    //=========================================================================
    // TRK_COMPLETE
    // Kết thúc một object; nếu Execute còn TRUE thì tìm object tiếp theo.
    //=========================================================================
    E_TrackingState.TRK_COMPLETE:

        // Chu trình một object đã hoàn thành.
		Runtime.Response.Busy := FALSE;
		Runtime.Response.Done := TRUE;
	
		// Giữ output ở trạng thái an toàn.
		VacuumCommand := FALSE;
		BlowCommand := FALSE;
	
		// Chỉ về IDLE khi tầng Command Engine hạ Execute.
		IF NOT Execute THEN
			Runtime.Response.Accepted := FALSE;
			Runtime.Response.Done := FALSE;
			Runtime.State := E_TrackingState.TRK_IDLE;
		END_IF;


    //=========================================================================
    // TRK_ABORT_ACTIVE
    // Hủy motion vì object vượt vùng trước khi VacuumOK.
    //=========================================================================
    E_TrackingState.TRK_ABORT_ACTIVE:

        // Tắt hút vì chưa giữ được vật.
        VacuumCommand := FALSE;

        // Tắt thổi.
        BlowCommand := FALSE;

        // Bật yêu cầu abort motion.
        MotionAbort := TRUE;

        // Khi Motion Manager xác nhận abort hoàn tất.
        IF MotionAbortDone THEN
            // Hạ yêu cầu abort.
            MotionAbort := FALSE;

            // Xóa trạng thái motion.
            xMotionIssued := FALSE;
            xMotionRequestPending := FALSE;
            xMotionActive := FALSE;

            // Nếu PCS không còn InUse thì có thể tắt tracking.
            IF NOT fbTrackBelt.InUse THEN
                xTrackExecute := FALSE;

                // Chuyển sang vị trí an toàn.
                Runtime.State := E_TrackingState.TRK_MOVE_SAFE;
            END_IF;
        END_IF;

    //=========================================================================
    // TRK_MOVE_SAFE
    // Đưa robot về LeavePos sau khi bỏ object.
    //=========================================================================
    E_TrackingState.TRK_MOVE_SAFE:

        // Tắt hút.
        VacuumCommand := FALSE;

        // Tạo request Move Safe.
        IF NOT xMotionIssued AND NOT xMotionRequestPending AND NOT xMotionActive THEN

            // Dùng LeavePos làm điểm an toàn.
            MotionTarget := Config.LeavePos;

            // Dùng thông số Leave.
            MotionSpeed := Config.Motion.Leave.Speed;

            MotionAcceleration := Config.Motion.Leave.Acceleration;

            MotionDeceleration := Config.Motion.Leave.Deceleration;

            MotionJerk := Config.Motion.Leave.Jerk;

            MotionBlendRadius := Config.Motion.Leave.BlendRadius;

            // Chạy trong hệ robot/base.
            MotionCoordSystem := E_AppCoordSystem.APP_COORD_ROBOT_BASE;

            // Mã lệnh MoveL.
            MotionCommand := 2;

            // Bật request pending.
            xMotionRequestPending := TRUE;

            // Đánh dấu đã tạo lệnh.
            xMotionIssued := TRUE;
        END_IF;

        // Adapter đã nhận request.
        IF MotionAccepted AND xMotionRequestPending THEN
            xMotionRequestPending := FALSE;
            xMotionActive := TRUE;
        END_IF;

        // Move Safe hoàn thành.
        IF MotionDone AND xMotionActive THEN
            xMotionActive := FALSE;
            xMotionIssued := FALSE;

            Runtime.State := E_TrackingState.TRK_RELEASE_OBJECT;

        // Move Safe lỗi.
        ELSIF MotionError AND xMotionActive THEN
            xMotionActive := FALSE;

            Runtime.Response.Error := TRUE;
            Runtime.Response.ErrorID := MotionErrorID;

            Runtime.State := E_TrackingState.TRK_ERROR;
        END_IF;

    //=========================================================================
    // TRK_RELEASE_OBJECT
    // Giải phóng object MISSED và tiếp tục object kế tiếp.
    //=========================================================================
    E_TrackingState.TRK_RELEASE_OBJECT:

        // Tắt hút.
        VacuumCommand := FALSE;

        // Chỉ release khi PCS không còn InUse.
        IF NOT fbTrackBelt.InUse THEN
            // Tắt tracking PCS.
            xTrackExecute := FALSE;

            // Kiểm tra index trước khi truy cập Queue.
            IF Runtime.SelectedObjectIndex >= 1 AND Runtime.SelectedObjectIndex <= GVL.C_MAX_TRACK_OBJECTS THEN

                // Giải phóng object.
                Queue.Objects[Runtime.SelectedObjectIndex].Reserved := FALSE;
            END_IF;

            // Giải phóng ActiveIndex.
            Queue.ActiveIndex := GVL.C_INVALID_INDEX;

            // Xóa object active trong Runtime.
            Runtime.SelectedObjectIndex := 0;
            Runtime.SelectedObjectID := 0;

            // Xóa thông tin PCS.
            Runtime.PCSInfo.Valid := FALSE;
            Runtime.PCSInfo.InUse := FALSE;

            // Xóa trạng thái tool.
            xVacuumCaptured := FALSE;

            // Xóa trạng thái motion.
            xMotionIssued := FALSE;
            xMotionRequestPending := FALSE;
            xMotionActive := FALSE;

            // Tiếp tục tìm object khác.
            Runtime.State := E_TrackingState.TRK_FIND_OBJECT;
        END_IF;

    //=========================================================================
    // TRK_ABORTING
    // Hủy toàn ứng dụng khi Execute bị hạ.
    //=========================================================================
    E_TrackingState.TRK_ABORTING:

        // Tắt hút.
        VacuumCommand := FALSE;

        // Tắt thổi.
        BlowCommand := FALSE;

        // Yêu cầu abort motion.
        MotionAbort := TRUE;

        // Nếu có object active thì đánh dấu ABORTED.
        IF Runtime.SelectedObjectIndex >= 1 AND Runtime.SelectedObjectIndex <= GVL.C_MAX_TRACK_OBJECTS THEN

            Queue.Objects[Runtime.SelectedObjectIndex].State := E_TrackingObjectState.OBJ_ABORTED;

            Queue.Objects[Runtime.SelectedObjectIndex].Reserved := FALSE;
        END_IF;

        // Khi abort motion xong và PCS không còn InUse.
        IF MotionAbortDone AND NOT fbTrackBelt.InUse THEN

            // Hạ abort.
            MotionAbort := FALSE;

            // Tắt tracking PCS.
            xTrackExecute := FALSE;

            // Giải phóng ActiveIndex.
            Queue.ActiveIndex := GVL.C_INVALID_INDEX;

            // Xóa object active.
            Runtime.SelectedObjectIndex := 0;
            Runtime.SelectedObjectID := 0;

            // Xóa Busy và Accepted.
            Runtime.Response.Busy := FALSE;
            Runtime.Response.Accepted := FALSE;

            // Về IDLE.
            Runtime.State := E_TrackingState.TRK_IDLE;
        END_IF;

    //=========================================================================
    // TRK_ERROR
    // Giữ lỗi để Application Manager/HMI đọc.
    //=========================================================================
    E_TrackingState.TRK_ERROR:

        // Manager không còn xử lý bình thường.
        Runtime.Response.Busy := FALSE;

        // Giữ cờ Error.
        Runtime.Response.Error := TRUE;

        // Tắt hút.
        VacuumCommand := FALSE;

        // Tắt thổi.
        BlowCommand := FALSE;

        // Yêu cầu abort motion.
        MotionAbort := TRUE;

        // Nếu có object active thì đánh dấu ERROR.
        IF Runtime.SelectedObjectIndex >= 1 AND Runtime.SelectedObjectIndex <= GVL.C_MAX_TRACK_OBJECTS THEN

            Queue.Objects[Runtime.SelectedObjectIndex].State := E_TrackingObjectState.OBJ_ERROR;

            Queue.Objects[Runtime.SelectedObjectIndex].Reserved := FALSE;
        END_IF;

        // Chỉ tắt tracking khi PCS không còn InUse.
        IF NOT fbTrackBelt.InUse THEN
            xTrackExecute := FALSE;
        END_IF;

    //=========================================================================
    // STATE KHÔNG HỢP LỆ
    //=========================================================================
    ELSE
        // Báo lỗi state không hợp lệ.
        Runtime.Response.Error := TRUE;

        // Mã lỗi nội bộ cho state không hợp lệ.
        Runtime.Response.ErrorID := 6999;

        // Chuyển về TRK_ERROR.
        Runtime.State := E_TrackingState.TRK_ERROR;

END_CASE;

END_FUNCTION_BLOCK

// Just_Motion_Control_x86_64_Linux_SM_WV/Application/FB_/TOOL/FB_ToolManager
FUNCTION_BLOCK FB_ToolManager
VAR_INPUT

    // Cho phép Tool Manager.
    Enable : BOOL;

    // Command hiện tại.
    Command : ST_ToolCommand;

    // Cấu hình Tool.
    Config : ST_ToolConfig;

END_VAR

VAR_IN_OUT

    // Runtime Status của Tool.
    Status : ST_ToolStatus;

END_VAR

VAR

    // Bắt cạnh lên của Execute.
    rtExecute : R_TRIG;

    // Lệnh Tool đang chạy.
    eActiveCommand : E_ToolCommandType;

    // Timer dùng khi không cấu hình DI.
    tonAction : TON;

    // Timer giới hạn thời gian lệnh Tool.
    tonTimeout : TON;

    // Timer xác nhận GripOK ổn định.
    tonConfirm : TON;

    // Điều kiện lệnh Tool hoàn thành.
    xActionOK : BOOL;

    // Giá trị DI đang kiểm tra.
    xFeedbackDI : BOOL;

    // Thời gian giả lập nếu không có Sensor.
    tAction : TIME;

    // Timeout của lệnh Tool.
    tTimeout : TIME;

END_VAR

(*
===============================================================================
FUNCTION BLOCK
    FB_ToolManager

DESCRIPTION
    Điều khiển một Tool độc lập.

SUPPORTED COMMANDS
    - DOWN
    - GRIP
    - UP
    - RELEASE

FEEDBACK RULE
    - Nếu DI Channel > 0:
          Dùng DI làm điều kiện hoàn thành.
    - Nếu DI Channel = 0:
          Dùng Timer cấu hình tương ứng.
    - Nếu UseUpDown = FALSE:
          DOWN và UP hoàn thành ngay.

IMPORTANT
    - Chỉ FB này được phép ghi request IO của Tool.
    - Interpreter không nên ghi trực tiếp vào các DO đã thuộc Tool.
===============================================================================
*)

//=============================================================================
// DEFAULT PULSE OUTPUTS
//=============================================================================
Status.Accepted := FALSE;
Status.Done := FALSE;


//=============================================================================
// COPY TOOL ID TO STATUS
//=============================================================================
Status.ToolID := Config.ToolID;


//=============================================================================
// RESET / DISABLE
//=============================================================================
IF NOT Enable OR Command.Reset THEN

    Status.Busy := FALSE;

    Status.Error := FALSE;
    Status.ErrorID := 0;

    Status.State :=
        E_ToolRuntimeState.IDLE;

    tonAction(IN := FALSE);
    tonTimeout(IN := FALSE);
    tonConfirm(IN := FALSE);

    RETURN;

END_IF;


//=============================================================================
// ABORT
//=============================================================================
IF Command.Abort THEN

    Status.Busy := FALSE;

    Status.Error := TRUE;
    Status.ErrorID := 9299;

    Status.State :=
        E_ToolRuntimeState.ERROR;

    RETURN;

END_IF;


//=============================================================================
// DETECT NEW COMMAND
//=============================================================================
rtExecute(CLK := Command.Execute);

IF rtExecute.Q AND NOT Status.Busy THEN

    // Lưu loại lệnh hiện tại.
    eActiveCommand :=
        Command.CommandType;

    // Handshake.
    Status.Accepted := TRUE;
    Status.Busy := TRUE;

    Status.Error := FALSE;
    Status.ErrorID := 0;

    Status.ResponseCommandID :=
        Command.CommandID;

    // Reset timer trước khi bắt đầu lệnh mới.
    tonAction(IN := FALSE);
    tonTimeout(IN := FALSE);
    tonConfirm(IN := FALSE);

    // Gán State runtime.
    CASE eActiveCommand OF

        E_ToolCommandType.DOWN:
            Status.State :=
                E_ToolRuntimeState.DOWNING;

        E_ToolCommandType.GRIP:
            Status.State :=
                E_ToolRuntimeState.GRIPPING;

        E_ToolCommandType.UP:
            Status.State :=
                E_ToolRuntimeState.UPPING;

        E_ToolCommandType.RELEASE:
            Status.State :=
                E_ToolRuntimeState.RELEASING;

        ELSE
            Status.Busy := FALSE;
            Status.Done := TRUE;

    END_CASE;

END_IF;


//=============================================================================
// NO ACTIVE COMMAND
//=============================================================================
IF NOT Status.Busy THEN
    RETURN;
END_IF;


//=============================================================================
// RESET LOCAL ACTION FLAGS
//=============================================================================
xActionOK := FALSE;
xFeedbackDI := FALSE;

tAction := T#0MS;
tTimeout := T#1S;


//=============================================================================
// EXECUTE ACTIVE COMMAND
//=============================================================================
CASE eActiveCommand OF


    //=========================================================================
    // ACTION: DOWN
    //=========================================================================
    E_ToolCommandType.DOWN:

        // Tool không có cơ cấu Up/Down.
        IF NOT Config.UseUpDown THEN

            xActionOK := TRUE;

        ELSE

            //-----------------------------------------------------------------
            // COMMAND DOWN OUTPUT
            //-----------------------------------------------------------------
			
			IF Config.IO.UseSingleUpDownDO THEN
				// Single DO: phat muc DOWN.
				IF Config.IO.UpDownDOChannel > 0 AND Config.IO.UpDownDOChannel <= GVL.C_MAX_DO THEN
					GVL.Y[Config.IO.UpDownDOChannel] := Config.IO.DownDOActiveLevel;
				END_IF;
			ELSE
				// Dual DO: bat Down, tat Up.
				IF Config.IO.DownDOChannel > 0 AND Config.IO.DownDOChannel <= GVL.C_MAX_DO THEN
					GVL.Y[Config.IO.DownDOChannel] := Config.IO.DownDOActiveLevel;
				END_IF;
			
				IF Config.IO.UpDOChannel > 0 AND Config.IO.UpDOChannel <= GVL.C_MAX_DO THEN
					GVL.Y[Config.IO.UpDOChannel] := NOT Config.IO.UpDOActiveLevel;
				END_IF;
			END_IF;


            //-----------------------------------------------------------------
            // CHECK DOWN FEEDBACK
            //-----------------------------------------------------------------
            IF Config.IO.DownOKDIChannel = 0 THEN

                // Không có DI -> dùng Timer.
                tAction :=
                    Config.DownTimeNoSensor;

                tonAction(
                    IN := TRUE,
                    PT := tAction
                );

                xActionOK :=
                    tonAction.Q;

            ELSE

                // Có DI -> dùng Sensor.
                xActionOK :=
                    GVL.X[
                        Config.IO.DownOKDIChannel
                    ] = Config.IO.DownOKDIActiveLevel;

            END_IF;


            // Timeout của DOWN.
            tTimeout :=
                Config.DownTimeout;

        END_IF;


    //=========================================================================
    // ACTION: GRIP
    //=========================================================================
    E_ToolCommandType.GRIP:

        //---------------------------------------------------------------------
        // RESET RELEASE OUTPUT
        //---------------------------------------------------------------------
        IF Config.IO.UseSingleGripReleaseDO THEN
			IF Config.IO.GripReleaseDOChannel > 0 AND Config.IO.GripReleaseDOChannel <= GVL.C_MAX_DO THEN
				GVL.Y[Config.IO.GripReleaseDOChannel] := Config.IO.GripDOActiveLevel;
			END_IF;
		ELSE
			IF Config.IO.ReleaseDOChannel > 0 AND Config.IO.ReleaseDOChannel <= GVL.C_MAX_DO THEN
				GVL.Y[Config.IO.ReleaseDOChannel] := NOT Config.IO.ReleaseDOActiveLevel;
			END_IF;
			IF Config.IO.GripDOChannel > 0 AND Config.IO.GripDOChannel <= GVL.C_MAX_DO THEN
				GVL.Y[Config.IO.GripDOChannel] := Config.IO.GripDOActiveLevel;
			END_IF;
		END_IF;


        //---------------------------------------------------------------------
        // CHECK GRIP FEEDBACK
        //---------------------------------------------------------------------
        IF Config.IO.GripOKDIChannel = 0 THEN

            // Không có GripOK DI -> dùng Timer.
            tAction :=
                Config.GripTimeNoSensor;

            tonAction(
                IN := TRUE,
                PT := tAction
            );

            xActionOK :=
                tonAction.Q;

        ELSE

            // Có GripOK DI.
            xFeedbackDI :=
                GVL.X[
                    Config.IO.GripOKDIChannel
                ] = Config.IO.GripOKDIActiveLevel;

            // Xác nhận tín hiệu ổn định.
            tonConfirm(
                IN := xFeedbackDI,
                PT := Config.GripConfirmDelay
            );

            xActionOK :=
                tonConfirm.Q;

        END_IF;


        // Timeout của GRIP.
        tTimeout :=
            Config.GripTimeout;


    //=========================================================================
    // ACTION: UP
    //=========================================================================
    E_ToolCommandType.UP:

        // Tool không có cơ cấu Up/Down.
        IF NOT Config.UseUpDown THEN

            xActionOK := TRUE;

        ELSE

            //-----------------------------------------------------------------
            // RESET DOWN OUTPUT
            //-----------------------------------------------------------------
			IF Config.IO.UseSingleUpDownDO THEN
				// Single DO: UP = dao muc DOWN.
				IF Config.IO.UpDownDOChannel > 0 AND Config.IO.UpDownDOChannel <= GVL.C_MAX_DO THEN
					GVL.Y[Config.IO.UpDownDOChannel] := NOT Config.IO.DownDOActiveLevel;
				END_IF;
			ELSE
				// Dual DO: tat Down, bat Up.
				IF Config.IO.DownDOChannel > 0 AND Config.IO.DownDOChannel <= GVL.C_MAX_DO THEN
					GVL.Y[Config.IO.DownDOChannel] := NOT Config.IO.DownDOActiveLevel;
				END_IF;
			
				IF Config.IO.UpDOChannel > 0 AND Config.IO.UpDOChannel <= GVL.C_MAX_DO THEN
					GVL.Y[Config.IO.UpDOChannel] := Config.IO.UpDOActiveLevel;
				END_IF;
			END_IF;


            //-----------------------------------------------------------------
            // CHECK UP FEEDBACK
            //-----------------------------------------------------------------
            IF Config.IO.UpOKDIChannel = 0 THEN

                // Không có DI -> dùng Timer.
                tAction :=
                    Config.UpTimeNoSensor;

                tonAction(
                    IN := TRUE,
                    PT := tAction
                );

                xActionOK :=
                    tonAction.Q;

            ELSE

                // Có DI -> dùng Sensor.
                xActionOK :=
                    GVL.X[
                        Config.IO.UpOKDIChannel
                    ] = Config.IO.UpOKDIActiveLevel;

            END_IF;


            // Timeout của UP.
            tTimeout :=
                Config.UpTimeout;

        END_IF;


    //=========================================================================
    // ACTION: RELEASE
    //=========================================================================
    E_ToolCommandType.RELEASE:

        //---------------------------------------------------------------------
        // RESET GRIP OUTPUT
        //---------------------------------------------------------------------
        IF Config.IO.UseSingleGripReleaseDO THEN
			IF Config.IO.GripReleaseDOChannel > 0 AND Config.IO.GripReleaseDOChannel <= GVL.C_MAX_DO THEN
				GVL.Y[Config.IO.GripReleaseDOChannel] := NOT Config.IO.GripDOActiveLevel;
			END_IF;
		ELSE
			IF Config.IO.GripDOChannel > 0 AND Config.IO.GripDOChannel <= GVL.C_MAX_DO THEN
				GVL.Y[Config.IO.GripDOChannel] := NOT Config.IO.GripDOActiveLevel;
			END_IF;
			IF Config.IO.ReleaseDOChannel > 0 AND Config.IO.ReleaseDOChannel <= GVL.C_MAX_DO THEN
				GVL.Y[Config.IO.ReleaseDOChannel] := Config.IO.ReleaseDOActiveLevel;
			END_IF;
		END_IF;


        //---------------------------------------------------------------------
        // RELEASE CURRENTLY USES TIMER
        //---------------------------------------------------------------------
        tAction :=
            Config.ReleaseTimeNoSensor;

        tonAction(
            IN := TRUE,
            PT := tAction
        );

        xActionOK :=
            tonAction.Q;


        // Timeout của RELEASE.
        tTimeout :=
            Config.ReleaseTimeout;

END_CASE;


//=============================================================================
// ACTION TIMEOUT
//=============================================================================
tonTimeout(
    IN := TRUE,
    PT := tTimeout
);


//=============================================================================
// COMMAND COMPLETE
//=============================================================================
IF xActionOK THEN

    // Reset timer.
    tonAction(IN := FALSE);
    tonTimeout(IN := FALSE);
    tonConfirm(IN := FALSE);

    // Hoàn thành Handshake.
    Status.Busy := FALSE;
    Status.Done := TRUE;

    Status.Error := FALSE;
    Status.ErrorID := 0;


    //-------------------------------------------------------------------------
    // UPDATE TOOL RUNTIME STATE
    //-------------------------------------------------------------------------
    CASE eActiveCommand OF

        E_ToolCommandType.DOWN:

            Status.State :=
                E_ToolRuntimeState.DOWN;


        E_ToolCommandType.GRIP:

            Status.State :=
                E_ToolRuntimeState.OCCUPIED;

            Status.Occupied :=
                TRUE;

            Status.HeldObjectID :=
                Command.ObjectID;

            Status.GripOK :=
                TRUE;


        E_ToolCommandType.UP:

            IF Status.Occupied THEN

                Status.State :=
                    E_ToolRuntimeState.OCCUPIED;

            ELSE

                Status.State :=
                    E_ToolRuntimeState.UP;

            END_IF;


        E_ToolCommandType.RELEASE:

            Status.State :=
                E_ToolRuntimeState.IDLE;

            Status.Occupied :=
                FALSE;

            Status.HeldObjectID :=
                0;

            Status.GripOK :=
                FALSE;

    END_CASE;


//=============================================================================
// COMMAND ERROR
//=============================================================================
ELSIF tonTimeout.Q THEN

    Status.Busy := FALSE;

    Status.Error := TRUE;

    // Mã lỗi được tạo từ loại lệnh Tool.
    Status.ErrorID :=
        9200 + TO_UDINT(eActiveCommand);

    Status.State :=
        E_ToolRuntimeState.ERROR;

END_IF;

END_FUNCTION_BLOCK

// Just_Motion_Control_x86_64_Linux_SM_WV/Application/FC_/TrackingQueue/F_SelectTrackingObject
FUNCTION F_SelectTrackingObject  : UINT
VAR_INPUT
    // Thuật toán lựa chọn object.
    SelectMode : E_TrackingSelectMode;

    // ObjectID được yêu cầu khi chọn theo ID cụ thể.
    SpecificID : UDINT;

    // Chiều chuyển động conveyor.
    // +1: tọa độ tăng.
    // -1: tọa độ giảm.
    DirectionSign : SINT;

    // Điểm Vision tối thiểu.
    MinimumVisionScore : REAL;

    // Queue cần tìm object.
    Queue : ST_TRACKING_QUEUE;
END_VAR
VAR
    // Index dùng duyệt toàn bộ Queue.
    uiIndex : UINT;

    // Index object tốt nhất đã tìm thấy.
    uiBestIndex : UINT;

    // TRUE sau khi đã tìm được ít nhất một candidate.
    xFoundCandidate : BOOL;

    // Giá trị so sánh REAL của object tốt nhất.
    rBestValue : REAL;

    // Giá trị so sánh UINT của object tốt nhất.
    uiBestPriority : UINT;

    // Thời điểm capture tốt nhất cho FIFO.
    tBestCaptureTime : TIME;

    // Object hiện tại trong vòng lặp.
    stCandidate : ST_TRACKING_OBJECT;
END_VAR

// Khởi tạo kết quả là index không hợp lệ.
uiBestIndex := GVL.C_INVALID_INDEX;

// Chưa có candidate nào được tìm thấy.
xFoundCandidate := FALSE;

// Khởi tạo biến so sánh.
rBestValue := 0.0;
uiBestPriority := 0;
tBestCaptureTime := T#0MS;


// Duyệt toàn bộ object trong Queue.
FOR uiIndex := 1 TO GVL.C_MAX_TRACK_OBJECTS DO

    // Lấy bản sao object hiện tại để code dễ đọc.
    stCandidate := Queue.Objects[uiIndex];

    // Chỉ tiếp tục nếu object đủ điều kiện tham gia Scheduler.
    IF F_IsTrackingObjectSelectable(
        TrackingObject := stCandidate,
        MinimumVisionScore := MinimumVisionScore
    ) THEN

        CASE SelectMode OF

            //===============================================================
            // Không tự động chọn object.
            //===============================================================
            E_TrackingSelectMode.TRACK_SELECT_NONE:

                // Không thay đổi uiBestIndex.
                ;


            //===============================================================
            // Chọn đúng ObjectID do Application yêu cầu.
            //===============================================================
            E_TrackingSelectMode.TRACK_SELECT_SPECIFIC_ID:

                IF stCandidate.ObjectID = SpecificID THEN
                    // Tìm đúng ObjectID thì trả về ngay.
                    F_SelectTrackingObject := uiIndex;
                    RETURN;
                END_IF;


            //===============================================================
            // FIFO: chọn object có CaptureTime nhỏ nhất.
            //===============================================================
            E_TrackingSelectMode.TRACK_SELECT_FIFO:

                IF NOT xFoundCandidate THEN
                    // Candidate đầu tiên tạm thời là tốt nhất.
                    uiBestIndex := uiIndex;
                    tBestCaptureTime := stCandidate.CaptureTime;
                    xFoundCandidate := TRUE;

                ELSIF stCandidate.CaptureTime < tBestCaptureTime THEN
                    // Object được ghi nhận sớm hơn sẽ được ưu tiên.
                    uiBestIndex := uiIndex;
                    tBestCaptureTime := stCandidate.CaptureTime;
                END_IF;


            //===============================================================
            // Chọn object gần điểm thoát nhất.
            //===============================================================
            E_TrackingSelectMode.TRACK_SELECT_NEAREST_EXIT:

                IF NOT xFoundCandidate THEN
                    // Candidate đầu tiên tạm thời là tốt nhất.
                    uiBestIndex := uiIndex;
                    rBestValue := stCandidate.ConveyorCoordinate;
                    xFoundCandidate := TRUE;

                ELSIF DirectionSign >= 0 THEN
                    // Conveyor chạy chiều tăng:
                    // tọa độ lớn hơn nghĩa là object đi trước hơn.
                    IF stCandidate.ConveyorCoordinate > rBestValue THEN
                        uiBestIndex := uiIndex;
                        rBestValue := stCandidate.ConveyorCoordinate;
                    END_IF;

                ELSE
                    // Conveyor chạy chiều giảm:
                    // tọa độ nhỏ hơn nghĩa là object đi trước hơn.
                    IF stCandidate.ConveyorCoordinate < rBestValue THEN
                        uiBestIndex := uiIndex;
                        rBestValue := stCandidate.ConveyorCoordinate;
                    END_IF;
                END_IF;


            //===============================================================
            // Earliest Deadline First:
            // chọn object có TimeRemainingSec nhỏ nhất.
            //===============================================================
            E_TrackingSelectMode.TRACK_SELECT_MIN_TIME_REMAIN:

                IF NOT xFoundCandidate THEN
                    // Candidate đầu tiên tạm thời là tốt nhất.
                    uiBestIndex := uiIndex;
                    rBestValue := stCandidate.TimeRemainingSec;
                    xFoundCandidate := TRUE;

                ELSIF stCandidate.TimeRemainingSec < rBestValue THEN
                    // Object còn ít thời gian hơn được ưu tiên.
                    uiBestIndex := uiIndex;
                    rBestValue := stCandidate.TimeRemainingSec;
                END_IF;


            //===============================================================
            // Chọn Priority lớn nhất.
            // Nếu bằng Priority thì chọn TimeRemainingSec nhỏ hơn.
            //===============================================================
            E_TrackingSelectMode.TRACK_SELECT_HIGHEST_PRIORITY:

                IF NOT xFoundCandidate THEN
                    // Candidate đầu tiên tạm thời là tốt nhất.
                    uiBestIndex := uiIndex;
                    uiBestPriority := stCandidate.Priority;
                    rBestValue := stCandidate.TimeRemainingSec;
                    xFoundCandidate := TRUE;

                ELSIF stCandidate.Priority > uiBestPriority THEN
                    // Priority lớn hơn thắng trực tiếp.
                    uiBestIndex := uiIndex;
                    uiBestPriority := stCandidate.Priority;
                    rBestValue := stCandidate.TimeRemainingSec;

                ELSIF (stCandidate.Priority = uiBestPriority)
                   AND (stCandidate.TimeRemainingSec < rBestValue) THEN
                    // Khi Priority bằng nhau, object gần deadline hơn thắng.
                    uiBestIndex := uiIndex;
                    rBestValue := stCandidate.TimeRemainingSec;
                END_IF;


            //===============================================================
            // Chọn VisionScore lớn nhất.
            // Nếu bằng VisionScore thì chọn TimeRemainingSec nhỏ hơn.
            //===============================================================
            E_TrackingSelectMode.TRACK_SELECT_HIGHEST_VISION_SCORE:

                IF NOT xFoundCandidate THEN
                    // Candidate đầu tiên tạm thời là tốt nhất.
                    uiBestIndex := uiIndex;
                    rBestValue := stCandidate.VisionScore;
                    xFoundCandidate := TRUE;

                ELSIF stCandidate.VisionScore > rBestValue THEN
                    // VisionScore cao hơn được ưu tiên.
                    uiBestIndex := uiIndex;
                    rBestValue := stCandidate.VisionScore;

                ELSIF stCandidate.VisionScore = rBestValue THEN
                    // Nếu score bằng nhau, dùng TimeRemainingSec làm tie-break.
                    IF stCandidate.TimeRemainingSec
                       < Queue.Objects[uiBestIndex].TimeRemainingSec THEN

                        uiBestIndex := uiIndex;
                    END_IF;
                END_IF;


            //===============================================================
            // Chọn thời gian gắp ước tính nhỏ nhất.
            //===============================================================
            E_TrackingSelectMode.TRACK_SELECT_SHORTEST_PICK_TIME:

                IF NOT xFoundCandidate THEN
                    // Candidate đầu tiên tạm thời là tốt nhất.
                    uiBestIndex := uiIndex;
                    rBestValue := stCandidate.EstimatedPickTimeSec;
                    xFoundCandidate := TRUE;

                ELSIF stCandidate.EstimatedPickTimeSec < rBestValue THEN
                    // Object có thời gian gắp ước tính ngắn hơn được ưu tiên.
                    uiBestIndex := uiIndex;
                    rBestValue := stCandidate.EstimatedPickTimeSec;
                END_IF;


            ELSE
                // SelectMode không hợp lệ:
                // không chọn object để tránh hành vi không xác định.
                ;

        END_CASE;

    END_IF;

END_FOR;

// Trả về index object được Scheduler chọn.
// Nếu không có object phù hợp, kết quả là C_INVALID_INDEX.
F_SelectTrackingObject := uiBestIndex;

END_FUNCTION

// Just_Motion_Control_x86_64_Linux_SM_WV/Application/FC_/Conveyor/F_IsTrackingObjectSelectable
FUNCTION F_IsTrackingObjectSelectable : BOOL
VAR_INPUT
    // Object cần kiểm tra.
    TrackingObject : ST_TRACKING_OBJECT;

    // Điểm Vision tối thiểu cho phép.
    MinimumVisionScore : REAL;
END_VAR

// Mặc định object không được phép chọn.
F_IsTrackingObjectSelectable := FALSE;

// Chỉ object hợp lệ mới được xét tiếp.
IF NOT TrackingObject.Valid THEN
    RETURN;
END_IF;

// Object đã Reserved không được Scheduler chọn lại.
IF TrackingObject.Reserved THEN
    RETURN;
END_IF;

// Chỉ object đã READY mới được chọn.
IF TrackingObject.State
   <> E_TrackingObjectState.OBJ_READY THEN
    RETURN;
END_IF;

// Object phải còn đủ điều kiện gắp.
IF NOT TrackingObject.CanPick THEN
    RETURN;
END_IF;

// Object có điểm Vision thấp hơn giới hạn thì bị loại.
IF TrackingObject.VisionScore < MinimumVisionScore THEN
    RETURN;
END_IF;

// Qua toàn bộ điều kiện thì object hợp lệ cho Scheduler.
F_IsTrackingObjectSelectable := TRUE;

END_FUNCTION

// Just_Motion_Control_x86_64_Linux_SM_WV/Application/FB_/ConveyorTrack/FB_MultiToolTrackingController_A
FUNCTION_BLOCK FB_MultiToolTrackingController_A
VAR_INPUT
    Command : ST_MultiToolTrackingCommand;
    CoreAccepted : BOOL;
    CoreBusy : BOOL;
    CoreSyncOK : BOOL;
    CorePCSInUse : BOOL;
    CoreReleased : BOOL;
    CoreError : BOOL;
    CoreErrorID : UDINT;
    SelectToolDone : BOOL;
    SelectToolError : BOOL;
    SelectToolErrorID : UDINT;
END_VAR
VAR_IN_OUT
    Queue : ST_TRACKING_QUEUE;
    ToolConfig : ARRAY[0..GVL.C_MAX_TOOLS] OF ST_ToolConfig;
    ToolStatus : ARRAY[0..GVL.C_MAX_TOOLS] OF ST_ToolStatus;
    Recipes : ARRAY[0..GVL.C_MAX_TRACK_RECIPES] OF ST_MultiToolTrackingRecipe;
    Status : ST_MultiToolTrackingStatus;
END_VAR
VAR_OUTPUT
    CoreStart : BOOL;
    CoreRelease : BOOL;
    CoreAbort : BOOL;
    CoreReset : BOOL;
    CoreObjectIndex : UINT;
    CoreToolID : UINT;
    CorePickOffset : ST_POS;
    CoreApproachHeight : REAL;
    ToolCommand : ST_ToolCommand;
    SelectToolExecute : BOOL;
    SelectToolID : UINT;
    SelectToolTCP : ST_POS;
	CoreUseUpDown : BOOL;
	CoreUpDownStroke : REAL;
	CorePickSurfaceHeightMM : REAL;
END_VAR
VAR
    rtExecute : R_TRIG;
    fbScheduler : FB_ToolObjectScheduler;
    stRecipe : ST_MultiToolTrackingRecipe;
    uiToolIndex : UINT;
    uiObjectIndex : UINT;
    uiTargetCount : UINT;
    dwToolMask : DWORD;
    udiToolCommandID : UDINT;
    xCommandIssued : BOOL;
	// TRUE sau khi Controller đã giữ CoreRelease ít nhất một vòng quét.
	// Ngăn CoreReleased cũ làm bỏ qua tín hiệu PickerSafe.
	xReleaseArmed : BOOL;
	udiLastAcceptedCommandID : UDINT := 0;
END_VAR

(*
===============================================================================
FB_MultiToolTrackingController_A

MỤC ĐÍCH
    Điều phối một lệnh TRACK_ON cho Robot A.

CHU TRÌNH
    IDLE
    -> LOAD_RECIPE
    -> SELECT_ASSIGNMENT
    -> SELECT_TOOL
    -> START_TRACKING
    -> WAIT_SYNC
    -> TOOL_DOWN
    -> TOOL_GRIP
    -> TOOL_UP
    -> RELEASE_TRACKING
    -> STORE_RESULT
    -> lặp đến khi đủ TargetPickCount
    -> COMPLETE

TRÁCH NHIỆM
    - Không gọi Motion trực tiếp.
    - Không gọi MC_TrackConveyorBelt trực tiếp.
    - Không ghi IO trực tiếp.
    - Chỉ điều phối Tracking Core, Tool Manager và Select Tool.
===============================================================================
*)
//=============================================================================
// DEFAULT PULSE OUTPUTS
//=============================================================================
Status.Accepted := FALSE;
Status.Done := FALSE;
CoreStart := FALSE;
CoreRelease := FALSE;
CoreAbort := FALSE;
CoreReset := FALSE;
ToolCommand.Execute := FALSE;
SelectToolExecute := FALSE;

//=============================================================================
// RESET
//=============================================================================
IF Command.Reset THEN
    Status.State := E_MultiTrackState.IDLE;
    Status.Busy := FALSE;
    Status.Error := FALSE;
    Status.ErrorID := 0;
    Status.PickedCount := 0;
    Status.SelectedToolID := 0;
    Status.SelectedObjectID := 0;
    CoreReset := TRUE;
    xCommandIssued := FALSE;
	xReleaseArmed := FALSE;
	udiLastAcceptedCommandID := 0;
    RETURN;
END_IF;

//=============================================================================
// ABORT
//=============================================================================
IF Command.Abort THEN 
	Status.State := E_MultiTrackState.ABORTING; 
	xReleaseArmed := FALSE;
END_IF;

// //=============================================================================
// // START COMMAND
// //=============================================================================
// rtExecute(CLK := Command.Execute);
// 
// IF rtExecute.Q AND Status.State = E_MultiTrackState.IDLE THEN
//     Status.Accepted := TRUE;
//     Status.Busy := TRUE;
//     Status.Error := FALSE;
//     Status.ErrorID := 0;
//     Status.ResponseCommandID := Command.CommandID;
//     Status.PickedCount := 0;
//     Status.OccupiedToolMask := 0;
//     Status.State := E_MultiTrackState.LOAD_RECIPE;
// END_IF;

//=============================================================================
// START NEW COMMAND
//-----------------------------------------------------------------------------
// Không phụ thuộc riêng cạnh Execute.
// CommandID là khóa transaction chính.
//=============================================================================
IF Command.Execute
AND Command.CommandID <> 0
AND Command.CommandID <> udiLastAcceptedCommandID
AND Status.State = E_MultiTrackState.IDLE THEN

    udiLastAcceptedCommandID := Command.CommandID;

    Status.Accepted := TRUE;
    Status.Busy := TRUE;
    Status.Error := FALSE;
    Status.ErrorID := 0;

    Status.ResponseCommandID := Command.CommandID;
    Status.PickedCount := 0;
    Status.OccupiedToolMask := 0;

    Status.State := E_MultiTrackState.LOAD_RECIPE;

END_IF;


//=============================================================================
// STATE MACHINE
//=============================================================================
CASE Status.State OF

    E_MultiTrackState.IDLE:
        Status.Busy := FALSE;

    //-------------------------------------------------------------------------
    // Đọc Recipe và áp dụng tham số Override từ Interpreter.
    //-------------------------------------------------------------------------
    E_MultiTrackState.LOAD_RECIPE:
        IF Command.RecipeID = 0 OR Command.RecipeID > 32 OR NOT Recipes[Command.RecipeID].Enable THEN
            Status.Error := TRUE;
            Status.ErrorID := 9401;
            Status.State := E_MultiTrackState.ERROR;
        ELSE
            stRecipe := Recipes[Command.RecipeID];
            Status.ActiveRecipeID := stRecipe.RecipeID;
            IF Command.TargetPickCountOverride > 0 THEN uiTargetCount := Command.TargetPickCountOverride; ELSE uiTargetCount := stRecipe.TargetPickCount; END_IF;
            IF Command.ToolMaskOverride <> 0 THEN dwToolMask := Command.ToolMaskOverride; ELSE dwToolMask := stRecipe.ToolEnableMask; END_IF;
            Status.TargetPickCount := uiTargetCount;
            Status.State := E_MultiTrackState.VALIDATE_TOOLS;
        END_IF;

    //-------------------------------------------------------------------------
    // Kiểm tra nhanh cấu hình trước khi chạy.
    //-------------------------------------------------------------------------
    E_MultiTrackState.VALIDATE_TOOLS:
        IF uiTargetCount = 0 OR dwToolMask = 0 THEN
            Status.Error := TRUE;
            Status.ErrorID := 9402;
            Status.State := E_MultiTrackState.ERROR;
        ELSE
            Status.State := E_MultiTrackState.SELECT_ASSIGNMENT;
        END_IF;

    //-------------------------------------------------------------------------
    // Tìm một Tool rảnh và một Object phù hợp.
    //-------------------------------------------------------------------------
    E_MultiTrackState.SELECT_ASSIGNMENT:

		fbScheduler(
			Execute := TRUE,
			Recipe := stRecipe,
			ToolMask := dwToolMask,
			Queue := Queue,
			ToolConfig := ToolConfig,
			ToolStatus := ToolStatus
		);
	
		IF fbScheduler.Done AND fbScheduler.Valid THEN
			uiToolIndex := fbScheduler.ToolIndex;
			uiObjectIndex := fbScheduler.ObjectIndex;
	
			// Controller chỉ ghi Tool được phân công.
			// Tracking Manager là khối duy nhất được Reserve Object.
			Queue.Objects[uiObjectIndex].ReservedToolID := ToolConfig[uiToolIndex].ToolID;
	
			Status.SelectedToolID := ToolConfig[uiToolIndex].ToolID;
			Status.SelectedObjectID := Queue.Objects[uiObjectIndex].ObjectID;
	
			xCommandIssued := FALSE;
			Status.State := E_MultiTrackState.SELECT_ROBOT_TOOL;
		END_IF;

		
	//-------------------------------------------------------------------------
	// Chọn TCP/Tool cho Robot A.
	//-------------------------------------------------------------------------
	E_MultiTrackState.SELECT_ROBOT_TOOL:
	
		SelectToolID := ToolConfig[uiToolIndex].ToolID;
		SelectToolTCP := ToolConfig[uiToolIndex].ToolTCP;
		SelectToolExecute := TRUE;
	
		IF SelectToolDone THEN
			SelectToolExecute := FALSE;
			xCommandIssued := FALSE;
			Status.State := E_MultiTrackState.START_TRACKING;
	
		ELSIF SelectToolError THEN
			SelectToolExecute := FALSE;
			Status.Error := TRUE;
			Status.ErrorID := SelectToolErrorID;
			Status.State := E_MultiTrackState.ERROR;
		END_IF;
	
	
    //-------------------------------------------------------------------------
    // Phát request tới Tracking Core.
    //-------------------------------------------------------------------------
    E_MultiTrackState.START_TRACKING:
        CoreObjectIndex := uiObjectIndex;
        CoreToolID := ToolConfig[uiToolIndex].ToolID;
        CorePickOffset := ToolConfig[uiToolIndex].PickOffset;
        CoreApproachHeight := ToolConfig[uiToolIndex].ApproachHeight;
		CorePickSurfaceHeightMM := stRecipe.PickSurfaceHeightMM;
        CoreUseUpDown := ToolConfig[uiToolIndex].UseUpDown;
        CoreUpDownStroke := ToolConfig[uiToolIndex].UpDownStroke;
        CoreStart := TRUE;

        IF CoreAccepted OR CoreBusy THEN
            Queue.Objects[uiObjectIndex].State := E_TrackingObjectState.OBJ_TRACKING;
            Status.State := E_MultiTrackState.WAIT_SYNC;

        ELSIF CoreError THEN
            Status.Error := TRUE;
            Status.ErrorID := CoreErrorID;
            Status.State := E_MultiTrackState.ERROR;
        END_IF;

    //-------------------------------------------------------------------------
    // Chờ Robot tới Approach trong PCS và PCS vẫn InUse.
    //-------------------------------------------------------------------------
    E_MultiTrackState.WAIT_SYNC:
        Status.TrackingSyncOK := CoreSyncOK;
        Status.PCSInUse := CorePCSInUse;

        IF CoreSyncOK AND CorePCSInUse THEN
            xCommandIssued := FALSE;

            IF ToolConfig[uiToolIndex].UseUpDown THEN
                Status.State := E_MultiTrackState.TOOL_DOWN;
            ELSE
                Status.State := E_MultiTrackState.TOOL_GRIP;
            END_IF;

        ELSIF CoreError THEN
            Status.Error := TRUE;
            Status.ErrorID := CoreErrorID;
            Status.State := E_MultiTrackState.ERROR;
        END_IF;


    //-------------------------------------------------------------------------
	// COMMAND TOOL DOWN
	//-------------------------------------------------------------------------
	E_MultiTrackState.TOOL_DOWN:
	
		udiToolCommandID := udiToolCommandID + 1;
	
		ToolCommand.CommandID := udiToolCommandID;
		ToolCommand.ToolID := ToolConfig[uiToolIndex].ToolID;
		ToolCommand.CommandType := E_ToolCommandType.DOWN;
		ToolCommand.ObjectID := Queue.Objects[uiObjectIndex].ObjectID;
		ToolCommand.Execute := TRUE;
	
		Status.State := E_MultiTrackState.WAIT_TOOL_DOWN;
	
	
	//-------------------------------------------------------------------------
	// WAIT TOOL DOWN
	//-------------------------------------------------------------------------
	E_MultiTrackState.WAIT_TOOL_DOWN:
	
		IF ToolStatus[uiToolIndex].Done
		AND ToolStatus[uiToolIndex].ResponseCommandID = udiToolCommandID THEN
	
			Status.State := E_MultiTrackState.TOOL_GRIP;
	
		ELSIF ToolStatus[uiToolIndex].Error THEN
	
			Status.Error := TRUE;
			Status.ErrorID := ToolStatus[uiToolIndex].ErrorID;
			Status.State := E_MultiTrackState.ERROR;
	
		END_IF;
	
	
	//-------------------------------------------------------------------------
	// COMMAND TOOL GRIP
	//-------------------------------------------------------------------------
	E_MultiTrackState.TOOL_GRIP:
	
		udiToolCommandID := udiToolCommandID + 1;
	
		ToolCommand.CommandID := udiToolCommandID;
		ToolCommand.ToolID := ToolConfig[uiToolIndex].ToolID;
		ToolCommand.CommandType := E_ToolCommandType.GRIP;
		ToolCommand.ObjectID := Queue.Objects[uiObjectIndex].ObjectID;
		ToolCommand.Execute := TRUE;
	
		Status.State := E_MultiTrackState.WAIT_TOOL_GRIP;
	
	
	//-------------------------------------------------------------------------
	// WAIT TOOL GRIP
	//-------------------------------------------------------------------------
	E_MultiTrackState.WAIT_TOOL_GRIP:
	
		 IF ToolStatus[uiToolIndex].Done
        AND ToolStatus[uiToolIndex].ResponseCommandID = udiToolCommandID THEN

            IF ToolConfig[uiToolIndex].UseUpDown THEN
                Status.State := E_MultiTrackState.TOOL_UP;
            ELSE
                Status.State := E_MultiTrackState.RELEASE_TRACKING;
            END_IF;

        ELSIF ToolStatus[uiToolIndex].Error THEN
            Status.Error := TRUE;
            Status.ErrorID := ToolStatus[uiToolIndex].ErrorID;
            Status.State := E_MultiTrackState.ERROR;
        END_IF;
	
	
	//-------------------------------------------------------------------------
	// COMMAND TOOL UP
	//-------------------------------------------------------------------------
	E_MultiTrackState.TOOL_UP:
	
		udiToolCommandID := udiToolCommandID + 1;
	
		ToolCommand.CommandID := udiToolCommandID;
		ToolCommand.ToolID := ToolConfig[uiToolIndex].ToolID;
		ToolCommand.CommandType := E_ToolCommandType.UP;
		ToolCommand.ObjectID := Queue.Objects[uiObjectIndex].ObjectID;
		ToolCommand.Execute := TRUE;
	
		Status.State := E_MultiTrackState.WAIT_TOOL_UP;
	
	
	//-------------------------------------------------------------------------
	// WAIT TOOL UP
	//-------------------------------------------------------------------------
	E_MultiTrackState.WAIT_TOOL_UP:
	
		IF ToolStatus[uiToolIndex].Done
			AND ToolStatus[uiToolIndex].ResponseCommandID = udiToolCommandID THEN
		
				// Chuẩn bị một chu trình Release mới.
				xReleaseArmed := FALSE;
		
				Status.State := E_MultiTrackState.RELEASE_TRACKING;
		
			ELSIF ToolStatus[uiToolIndex].Error THEN
		
				Status.Error := TRUE;
				Status.ErrorID := ToolStatus[uiToolIndex].ErrorID;
				Status.State := E_MultiTrackState.ERROR;
		
			END_IF;

    //-------------------------------------------------------------------------
	// Báo PickerSafe để Tracking Core chạy Exit/Release PCS.
	//-------------------------------------------------------------------------
	E_MultiTrackState.RELEASE_TRACKING:
	
		// Phải giữ TRUE liên tục để Core Interface nhận được yêu cầu.
		CoreRelease := TRUE;
	
		// Vòng quét đầu tiên chỉ phát yêu cầu Release.
		// Không kiểm tra CoreReleased trong cùng vòng quét này.
		IF NOT xReleaseArmed THEN
	
			xReleaseArmed := TRUE;
	
		ELSE
	
			// Chỉ chấp nhận Released sau khi CoreRelease
			// đã được giữ ít nhất một vòng quét.
			IF CoreReleased THEN
	
				xReleaseArmed := FALSE;
				Status.State := E_MultiTrackState.STORE_RESULT;
	
			ELSIF CoreError THEN
	
				xReleaseArmed := FALSE;
				Status.Error := TRUE;
				Status.ErrorID := CoreErrorID;
				Status.State := E_MultiTrackState.ERROR;
				xReleaseArmed := FALSE;
			END_IF;
	
		END_IF;

    //-------------------------------------------------------------------------
    // Lưu kết quả Pick của Tool hiện tại.
    //-------------------------------------------------------------------------
    E_MultiTrackState.STORE_RESULT:
        Queue.Objects[uiObjectIndex].Reserved := FALSE;
        Queue.Objects[uiObjectIndex].State := E_TrackingObjectState.OBJ_PICKED;
        Status.PickedCount := Status.PickedCount + 1;
        Status.OccupiedToolMask := Status.OccupiedToolMask OR SHL(DWORD#1, uiToolIndex - 1);
        Status.State := E_MultiTrackState.CHECK_COUNT;

    //-------------------------------------------------------------------------
    // Đủ số lượng thì Done; chưa đủ thì chọn Tool/Object tiếp theo.
    //-------------------------------------------------------------------------
    E_MultiTrackState.CHECK_COUNT:
        IF Status.PickedCount >= uiTargetCount THEN
            Status.State := E_MultiTrackState.COMPLETE;
        ELSE
            Status.SelectedToolID := 0;
            Status.SelectedObjectID := 0;
            Status.TrackingSyncOK := FALSE;
            Status.PCSInUse := FALSE;
            Status.State := E_MultiTrackState.SELECT_ASSIGNMENT;
        END_IF;

    E_MultiTrackState.COMPLETE:
        Status.Busy := FALSE;
        Status.Done := TRUE;
        IF NOT Command.Execute THEN Status.State := E_MultiTrackState.IDLE; END_IF;

    E_MultiTrackState.ABORTING:
        CoreAbort := TRUE;
        Status.Busy := FALSE;
        Status.Error := TRUE;
        Status.ErrorID := 9499;
        Status.State := E_MultiTrackState.ERROR;

    E_MultiTrackState.ERROR:
        Status.Busy := FALSE;
        Status.Error := TRUE;
        IF NOT Command.Execute THEN Status.State := E_MultiTrackState.IDLE; END_IF;

END_CASE;

END_FUNCTION_BLOCK

// Just_Motion_Control_x86_64_Linux_SM_WV/Application/FB_/TOOL/FB_ToolObjectScheduler
FUNCTION_BLOCK FB_ToolObjectScheduler
VAR_INPUT

    // Bật thực hiện tìm Assignment.
    Execute : BOOL;

    // Recipe hiện tại.
    Recipe : ST_MultiToolTrackingRecipe;

    // Bitmask Tool được phép dùng.
    ToolMask : DWORD;

END_VAR

VAR_IN_OUT

    // Object Queue.
    Queue : ST_TRACKING_QUEUE;

    // Cấu hình Tool.
    ToolConfig : ARRAY[0..GVL.C_MAX_TOOLS] OF ST_ToolConfig;

    // Runtime Tool.
    ToolStatus : ARRAY[0..GVL.C_MAX_TOOLS] OF ST_ToolStatus;

END_VAR

VAR_OUTPUT

    // Tìm kiếm hoàn thành.
    Done : BOOL;

    // TRUE nếu tìm được cặp Tool - Object.
    Valid : BOOL;

    // Index Tool trong mảng.
    ToolIndex : UINT;

    // Index Object trong Queue.
    ObjectIndex : UINT;

END_VAR

VAR

    // Biến vòng lặp Tool.
    uiTool : UINT;

    // Biến vòng lặp Object.
    uiObject : UINT;

    // TRUE nếu Tool nằm trong Mask.
    xToolEnabledByMask : BOOL;

    // TRUE nếu ProductClass phù hợp.
    xProductClassValid : BOOL;
	xSourceValid : BOOL;
END_VAR

(*
===============================================================================
FUNCTION BLOCK
    FB_ToolObjectScheduler

DESCRIPTION
    Chọn một Tool đang rảnh và một Object hợp lệ.

SELECTION RULE
    1. Tool nằm trong ToolMask.
    2. Tool Enable và AllowTracking.
    3. Tool không Busy, không Occupied, không Error.
    4. Object Valid, CanPick, chưa Reserved.
    5. Object ở trạng thái OBJ_READY.
    6. ProductClass phù hợp Recipe và Tool.
===============================================================================
*)

//=============================================================================
// DEFAULT OUTPUT
//=============================================================================
Done := FALSE;
Valid := FALSE;
ToolIndex := 0;
ObjectIndex := 0;

//=============================================================================
// DISABLED
//=============================================================================
IF NOT Execute THEN RETURN; END_IF;

//=============================================================================
// SEARCH TOOL AND OBJECT
//=============================================================================
FOR uiTool := 1 TO GVL.C_MAX_TOOLS DO

    // Kiểm tra Tool có nằm trong ToolMask hay không.
    xToolEnabledByMask := (ToolMask AND SHL(DWORD#1, uiTool - 1)) <> 0;
	

    // Chỉ kiểm tra Object khi Tool sẵn sàng.
    IF xToolEnabledByMask
    AND ToolConfig[uiTool].Enable
    AND ToolConfig[uiTool].AllowTracking
    AND NOT ToolStatus[uiTool].Occupied
    AND NOT ToolStatus[uiTool].Busy
    AND NOT ToolStatus[uiTool].Error THEN

        FOR uiObject := 1 TO GVL.C_MAX_TRACK_OBJECTS DO

            // Kiểm tra Product Class phù hợp Recipe và Tool.
            xProductClassValid := (Recipe.ProductClassID = 0 OR Recipe.ProductClassID = Queue.Objects[uiObject].ProductClassID)
            AND (ToolConfig[uiTool].AllowedProductClassID = 0 OR ToolConfig[uiTool].AllowedProductClassID = Queue.Objects[uiObject].ProductClassID);
			
			// Kiểm tra Source phù hợp Recipe.
			xSourceValid := FALSE;
			
			CASE Recipe.ObjectSourceType OF
			
				E_ObjectSourceType.SENSOR:
					xSourceValid :=
						Queue.Objects[uiObject].SourceType = E_ObjectSourceType.SENSOR
						AND Queue.Objects[uiObject].SourceID = Recipe.SensorSourceID;
		
				E_ObjectSourceType.VISION:

					xSourceValid :=
						Queue.Objects[uiObject].SourceType =
							E_ObjectSourceType.VISION
				
						AND (
							(Recipe.VisionSourceID = 0)
							OR
							(Queue.Objects[uiObject].SourceID =
								Recipe.VisionSourceID)
						)
				
						AND Queue.Objects[uiObject].JobID =
							Recipe.VisionJobID;
							
// 				E_ObjectSourceType.VISION:
// 					xSourceValid :=
// 						Queue.Objects[uiObject].SourceType = E_ObjectSourceType.VISION
// 						AND Queue.Objects[uiObject].JobID = Recipe.VisionJobID;
			
				E_ObjectSourceType.NONE:
					// Giữ tương thích với bài test cũ.
					xSourceValid := TRUE;
			
			END_CASE;

	
            // Object phải hợp lệ, sẵn sàng gắp và chưa bị module khác giữ.
            IF Queue.Objects[uiObject].Valid
			AND Queue.Objects[uiObject].CanPick
			AND Queue.Objects[uiObject].State = E_TrackingObjectState.OBJ_READY
			AND NOT Queue.Objects[uiObject].Reserved
			AND xProductClassValid
			AND xSourceValid THEN

                ToolIndex := uiTool;
                ObjectIndex := uiObject;
                Valid := TRUE;
                Done := TRUE;
                RETURN;
            END_IF;

        END_FOR;

    END_IF;

END_FOR;

// Không tìm thấy cặp Tool/Object phù hợp.
Done := TRUE;

END_FUNCTION_BLOCK

// Just_Motion_Control_x86_64_Linux_SM_WV/Application/FB_/ConveyorTrack/FB_TrackingMotionQueueAdapter
FUNCTION_BLOCK FB_TrackingMotionQueueAdapter
VAR_INPUT
    Enable : BOOL;
    Reset : BOOL;

    Request : BOOL;
    Abort : BOOL;

    Target : ST_POS;
    Speed : REAL;
    Acceleration : REAL;
    Deceleration : REAL;
    Jerk : REAL;
    BlendRadius : REAL;
    CoordSystem : E_AppCoordSystem;
    Command : UINT;

    // Logic-only simulation không push vào robot.
    LogicSimulation : BOOL;
    LogicMotionDuration : TIME := T#300MS;
END_VAR

VAR_OUTPUT
    Accepted : BOOL;
    Busy : BOOL;
    Done : BOOL;
    Error : BOOL;
    ErrorID : UDINT;
    AbortDone : BOOL;
END_VAR

VAR
    fbPush : FB_MotionQueuePush;
    rtRequest : R_TRIG;
    tonLogicMotion : TON;

    stItem : ST_MotionQueueItem;
    xPushExecute : BOOL;
    xWaitingMotionResult : BOOL;
    xAcceptedLatched : BOOL;

    diRequestSequence : DINT := -1000;
    iActiveSourceStep : INT;
END_VAR

Accepted := FALSE;
Done := FALSE;
AbortDone := FALSE;

// Error không nên giữ từ request cũ khi Adapter đang không chờ motion.
IF NOT xPushExecute AND NOT xWaitingMotionResult THEN
    Error := FALSE;
    ErrorID := 0;
END_IF;

// IF Reset OR NOT Enable THEN
//     xPushExecute := FALSE;
//     xWaitingMotionResult := FALSE;
//     xAcceptedLatched := FALSE;
//     Busy := FALSE;
//     Error := FALSE;
//     ErrorID := 0;
//     tonLogicMotion(IN := FALSE);
//     fbPush(Execute := FALSE, Item := stItem);
//     RETURN;
// END_IF;

IF Reset OR NOT Enable THEN

    // Hạ yêu cầu push vào Motion Queue.
    xPushExecute := FALSE;

    // Không còn chờ kết quả motion trước.
    xWaitingMotionResult := FALSE;

    // Xóa cờ Accepted nội bộ.
    xAcceptedLatched := FALSE;

    // Xóa trạng thái output.
    Accepted := FALSE;
    Busy := FALSE;
    Done := FALSE;
    Error := FALSE;
    ErrorID := 0;
    AbortDone := FALSE;

    // Xóa SourceStep của request cũ.
    iActiveSourceStep := 0;

    // Hạ yêu cầu Abort còn sót lại.
    GVL.A_MotionAbortReq := FALSE;

    // Reset timer mô phỏng.
    tonLogicMotion(IN := FALSE);

    // Reset FB Push Motion Queue.
    fbPush(Execute := FALSE, Item := stItem);

    RETURN;
END_IF;

IF Abort THEN
    IF LogicSimulation THEN
        xWaitingMotionResult := FALSE;
        Busy := FALSE;
        AbortDone := TRUE;
    ELSE
        GVL.A_MotionAbortReq := TRUE;
        IF GVL.A_MotionAbortDone THEN
            GVL.A_MotionAbortReq := FALSE;
            xWaitingMotionResult := FALSE;
            Busy := FALSE;
            AbortDone := TRUE;
        END_IF;
    END_IF;
    RETURN;
END_IF;

rtRequest(CLK := Request);

//=============================================================================
// LOGIC-ONLY SIMULATION
//=============================================================================
IF LogicSimulation THEN
    IF rtRequest.Q AND NOT Busy THEN
        Accepted := TRUE;
        Busy := TRUE;
        tonLogicMotion(IN := FALSE);
    END_IF;

    tonLogicMotion(IN := Busy, PT := LogicMotionDuration);

    IF tonLogicMotion.Q THEN
        tonLogicMotion(IN := FALSE);
        Busy := FALSE;
        Done := TRUE;
    END_IF;

    RETURN;
END_IF;

//=============================================================================
// ROBOT REAL: ĐÓNG GÓI VÀ PUSH VÀO MOTION QUEUE ROBOT A
//=============================================================================
IF rtRequest.Q AND NOT xPushExecute AND NOT xWaitingMotionResult THEN
    diRequestSequence := diRequestSequence - 1;
    IF diRequestSequence < -30000 THEN diRequestSequence := -1000; END_IF;
    iActiveSourceStep := DINT_TO_INT(diRequestSequence);

    stItem.Cmd := E_RobotCmd.CMD_MovL;
    stItem.SourceStep := iActiveSourceStep;
    stItem.PointNo := 0;
    stItem.MidPointNo := 0;
    stItem.EndPointNo := 0;
    stItem.Speed := REAL_TO_LREAL(Speed);
    stItem.BlendMode := GVL.C_TM_None;
    stItem.BlendRadius := REAL_TO_LREAL(BlendRadius);
    stItem.CircleMode := 0;
    stItem.PathChoice := 0;
    stItem.SkipPositionCheck := TRUE;

    stItem.UseDirectPosition := TRUE;
    stItem.DirectPosition := Target;
    stItem.DirectCoordSystem := F_MapAppCoordSystem(Coord := CoordSystem);
    stItem.Acceleration := REAL_TO_LREAL(Acceleration);
    stItem.Deceleration := REAL_TO_LREAL(Deceleration);
    stItem.Jerk := REAL_TO_LREAL(Jerk);
    stItem.ApplicationCommandID := TO_UDINT(ABS(iActiveSourceStep));

    xPushExecute := TRUE;
END_IF;

fbPush(Execute := xPushExecute, Item := stItem);

IF xPushExecute AND fbPush.Done THEN
    xPushExecute := FALSE;
    xWaitingMotionResult := TRUE;
    xAcceptedLatched := TRUE;
    Accepted := TRUE;
    Busy := TRUE;
END_IF;

IF xPushExecute AND fbPush.Error THEN
    xPushExecute := FALSE;
    Error := TRUE;
    ErrorID := 7201; // Motion Queue full / Push failed.
END_IF;

// Reset handshake của FB Push sau khi push xong.
IF NOT xPushExecute THEN fbPush(Execute := FALSE, Item := stItem); END_IF;

// Theo dõi đúng item bằng SourceStep âm riêng của Application.
IF xWaitingMotionResult THEN
    Busy := TRUE;

//     IF GVL.A_MotionDonePulse AND GVL.A_MotionDoneStep = iActiveSourceStep THEN
//         xWaitingMotionResult := FALSE;
//         Busy := FALSE;
//         Done := TRUE;
//     END_IF;
// 
//     IF GVL.A_MotionErrorPulse AND GVL.A_MotionErrorStep = iActiveSourceStep THEN
//         xWaitingMotionResult := FALSE;
//         Busy := FALSE;
//         Error := TRUE;
//         ErrorID := INT_TO_UDINT(GVL.A_MotionErrorCode);
//     END_IF;
	
	IF GVL.A_MotionDonePulse AND GVL.A_MotionDoneStep = iActiveSourceStep THEN
		xWaitingMotionResult := FALSE;
		xAcceptedLatched := FALSE;
		Busy := FALSE;
		Done := TRUE;
	END_IF;
	
	// Motion hiện tại báo lỗi đúng SourceStep.
	IF GVL.A_MotionErrorPulse AND GVL.A_MotionErrorStep = iActiveSourceStep THEN
		xWaitingMotionResult := FALSE;
		xAcceptedLatched := FALSE;
		Busy := FALSE;
		Error := TRUE;
		ErrorID := INT_TO_UDINT(GVL.A_MotionErrorCode);
	END_IF;
END_IF;

END_FUNCTION_BLOCK

// Just_Motion_Control_x86_64_Linux_SM_WV/Application/FC_/Coordinate_TF/F_MapAppCoordSystem
FUNCTION F_MapAppCoordSystem : SMC_COORD_SYSTEM
VAR_INPUT
    Coord : E_AppCoordSystem;
END_VAR

//=============================================================================
// F_MapAppCoordSystem
//-----------------------------------------------------------------------------
// Chuyển hệ tọa độ của Application sang hệ tọa độ SoftMotion.
//=============================================================================

CASE Coord OF

    // Robot Base phải ánh xạ sang MCS.
    E_AppCoordSystem.APP_COORD_ROBOT_BASE:
        F_MapAppCoordSystem := SMC_COORD_SYSTEM.MCS;

    // Conveyor Tracking số 1.
    E_AppCoordSystem.APP_COORD_PCS1:
        F_MapAppCoordSystem := SMC_COORD_SYSTEM.PCS_1;

    // Nếu có PCS_2.
    E_AppCoordSystem.APP_COORD_PCS2:
        F_MapAppCoordSystem := SMC_COORD_SYSTEM.PCS_2;

    ELSE
        // Không nên mặc định về PCS_1.
        // Khi không xác định, dùng Robot Base an toàn hơn.
        F_MapAppCoordSystem := SMC_COORD_SYSTEM.MCS;

END_CASE;

END_FUNCTION

// Just_Motion_Control_x86_64_Linux_SM_WV/Application/PRG_ROBOT/PRG_TrackingObjectSource_B
PROGRAM PRG_TrackingObjectSource_B
VAR
    fbSensorSourceB : ARRAY[1..GVL.C_MAX_SENSOR_SOURCES] OF FB_SensorObjectSource; // Biến nội bộ fbSensorSourceB.
    uiSensorSource : UINT; // Biến nội bộ uiSensorSource.
    fbVisionSourceB : ARRAY[1..GVL.C_MAX_VISION_CHANNELS] OF FB_VisionObjectSource; // Biến nội bộ fbVisionSourceB.
    uiVisionSource : UINT; // Biến nội bộ uiVisionSource.
    fbVisionResultAdapterB : ARRAY[1..GVL.C_MAX_VISION_CHANNELS] OF FB_VisionTrackingResultAdapter; // Biến nội bộ fbVisionResultAdapterB.
    fbVisionTriggerB : ARRAY[1..GVL.C_MAX_VISION_CHANNELS] OF FB_VisionTrackingTrigger; // Mỗi Vision Source có một Trigger FB độc lập để giữ TriggerID và pitch riêng.
    uiCamera : UINT; // Camera đang xử lý trong loop.
    uiTrackingRecipe : UINT; // Recipe TRACK_PICK hiện tại.
    xTrackingVisionEnable : BOOL; // TRUE khi Recipe/Command hiện tại cho phép Source này trigger nền.
    xVisionCommandAccepted : BOOL; // TRUE khi Vision Framework đã nhận đúng TriggerID đang chờ.
END_VAR

//=============================================================================
// PRG_TrackingObjectSource_A
//-----------------------------------------------------------------------------
// Quản lý nhiều Sensor Source cho Tracking Queue Robot A.
// Mỗi Sensor Source có một FB riêng để giữ debounce, edge và spacing riêng.
//=============================================================================

//=============================================================================
// 1. SENSOR OBJECT SOURCES
//=============================================================================
FOR uiSensorSource := 1 TO GVL.C_MAX_SENSOR_SOURCES DO

    fbSensorSourceB[uiSensorSource](
        Enable := GVL.g_aSensorSourceConfigB[uiSensorSource].Enable,
        Reset := GVL.g_xResetTrackingObjectSourceB,
        Config := GVL.g_aSensorSourceConfigB[uiSensorSource],
        ConveyorPositionMM := REAL_TO_LREAL(GVL.g_aConveyorRuntime[2].Status.PositionMM),
        Queue := GVL.g_stTrackingQueue_B
    );

END_FOR;


//=============================================================================
// 2. VISION TRACKING BACKGROUND TRIGGER
//-----------------------------------------------------------------------------
// TRACK_PICK đang Execute sẽ mở Tracking Session.
// Chỉ Source có VisionSourceID đúng với Recipe đang chạy mới được trigger.
//=============================================================================
FOR uiVisionSource := 1 TO GVL.C_MAX_VISION_CHANNELS DO

    uiCamera := GVL.g_aVisionTrackingSourceConfigB[uiVisionSource].CameraID;
    uiTrackingRecipe := GVL.g_stMultiTrackCommandB.RecipeID;

    // Mặc định Source không được trigger.
    xTrackingVisionEnable := FALSE;

    // Chỉ bật nếu Recipe hợp lệ, command TRACK_PICK đang active và Recipe dùng Vision Source này.
    IF GVL.g_stMultiTrackCommandB.Execute
    AND uiTrackingRecipe > 0
    AND uiTrackingRecipe <= GVL.C_MAX_TRACK_RECIPES
    AND GVL.g_aMultiTrackRecipeB[uiTrackingRecipe].Enable
    AND GVL.g_aMultiTrackRecipeB[uiTrackingRecipe].ObjectSourceType = E_ObjectSourceType.VISION
    AND GVL.g_aMultiTrackRecipeB[uiTrackingRecipe].VisionSourceID = GVL.g_aVisionTrackingSourceConfigB[uiVisionSource].VisionSourceID THEN
        xTrackingVisionEnable := GVL.g_aVisionTrackingSourceConfigB[uiVisionSource].Enable;
    //END_IF;
	// Commissioning: chỉ mở Source 1 mà chưa cần TRACK_PICK.
	ELSIF GVL.g_xVisionTrackingAutoTriggerTestB AND uiVisionSource = 1 THEN
		xTrackingVisionEnable := GVL.g_aVisionTrackingSourceConfigB[uiVisionSource].Enable;
	END_IF;

    // CameraID phải hợp lệ trước khi đọc g_aVisionStatus[].
    IF xTrackingVisionEnable AND uiCamera > 0 AND uiCamera <= GVL.C_MAX_VISION_CHANNELS THEN

        // Vision xác nhận command khi CurrentTriggerID bằng TriggerID đang chờ.
        xVisionCommandAccepted := fbVisionTriggerB[uiVisionSource].WaitingAccepted
            AND GVL.g_aVisionStatus[uiCamera].CurrentTriggerID = fbVisionTriggerB[uiVisionSource].TriggerID;

        fbVisionTriggerB[uiVisionSource](
            Enable := TRUE,
            Reset := GVL.g_xResetTrackingObjectSourceB,
            Config := GVL.g_aVisionTrackingSourceConfigB[uiVisionSource],
            ConveyorPositionMM := REAL_TO_LREAL(GVL.g_aConveyorRuntime[2].Status.PositionMM),

            // TODO:
            // Thay 0.0 bằng field Velocity thực tế của ST_CONVEYOR_STATUS sau khi anh chốt tên field.
            // Trong thời gian test có thể đặt TriggerOnlyWhenMoving = FALSE.
            ConveyorVelocityMMs := GVL.g_aConveyorRuntime[2].Status.VelocityMMs,

            VisionReady := GVL.g_aVisionStatus[uiCamera].Ready,
            VisionBusy := GVL.g_aVisionStatus[uiCamera].Busy,
            CommandAccepted := xVisionCommandAccepted,
			ResultProcessedTriggerID := fbVisionSourceB[uiVisionSource].LastProcessedTriggerID
        );

        //---------------------------------------------------------------------
        // MAP TRACKING TRIGGER -> VISION COMMAND
        //---------------------------------------------------------------------
        // Execute được giữ TRUE tới khi CurrentTriggerID xác nhận đã nhận command,
        // nên Communication task 15 ms không bỏ lỡ request từ task 4 ms.
        IF fbVisionTriggerB[uiVisionSource].TriggerExecute THEN
            GVL.g_aVisionCommand[uiCamera].CameraID := uiCamera;
            GVL.g_aVisionCommand[uiCamera].JobID := GVL.g_aVisionTrackingSourceConfigB[uiVisionSource].JobID;
            GVL.g_aVisionCommand[uiCamera].Application := E_VisionApplication.VIS_APP_CONVEYOR_PICK;
            GVL.g_aVisionCommand[uiCamera].TriggerID := fbVisionTriggerB[uiVisionSource].TriggerID;
            GVL.g_aVisionCommand[uiCamera].ProductID := 0;
            GVL.g_aVisionCommand[uiCamera].CaptureConveyorPos := LREAL_TO_REAL(fbVisionTriggerB[uiVisionSource].CaptureConveyorPositionMM);
            GVL.g_aVisionCommand[uiCamera].Execute := TRUE;

        // Chỉ hạ Execute của command Tracking do chính Source này phát.
        ELSIF GVL.g_aVisionCommand[uiCamera].Application = E_VisionApplication.VIS_APP_CONVEYOR_PICK
        AND GVL.g_aVisionCommand[uiCamera].JobID = GVL.g_aVisionTrackingSourceConfigB[uiVisionSource].JobID THEN
            GVL.g_aVisionCommand[uiCamera].Execute := FALSE;
        END_IF;

    ELSE
        // Khi Source không active, reset FB để lần TRACK_PICK sau có thể trigger frame đầu ngay.
        fbVisionTriggerB[uiVisionSource](
            Enable := FALSE,
            Reset := GVL.g_xResetTrackingObjectSourceB,
            Config := GVL.g_aVisionTrackingSourceConfigB[uiVisionSource],
            ConveyorPositionMM := REAL_TO_LREAL(GVL.g_aConveyorRuntime[2].Status.PositionMM),
            ConveyorVelocityMMs := GVL.g_aConveyorRuntime[2].Status.VelocityMMs,
            VisionReady := FALSE,
            VisionBusy := FALSE,
            CommandAccepted := FALSE
        );
    END_IF;

END_FOR;


//=============================================================================
// 3. VISION RESULT ADAPTER
//-----------------------------------------------------------------------------
// Chuyển Result chung của Vision Framework thành Multi Result cho Tracking.
//=============================================================================
FOR uiVisionSource := 1 TO GVL.C_MAX_VISION_CHANNELS DO

    uiCamera := GVL.g_aVisionTrackingSourceConfigB[uiVisionSource].CameraID;

    IF uiCamera > 0 AND uiCamera <= GVL.C_MAX_VISION_CHANNELS THEN
        fbVisionResultAdapterB[uiVisionSource](
            Enable := GVL.g_aVisionTrackingSourceConfigB[uiVisionSource].Enable,
            Reset := GVL.g_xResetTrackingObjectSourceB,
            CameraID := uiCamera,
            JobID := GVL.g_aVisionTrackingSourceConfigB[uiVisionSource].JobID,
            VisionResult := GVL.g_aVisionResult[uiCamera]
        );

        // Lưu Multi Result chuẩn để Vision Object Source xử lý ở bước tiếp theo.
        GVL.g_aVisionTrackingMultiResultB[uiVisionSource] := fbVisionResultAdapterB[uiVisionSource].TrackingResult;
    END_IF;

END_FOR;


//=============================================================================
// 4. VISION OBJECT SOURCES
//-----------------------------------------------------------------------------
// Scale/Offset -> Duplicate Check -> Push Object mới vào Tracking Queue.
//=============================================================================
FOR uiVisionSource := 1 TO GVL.C_MAX_VISION_CHANNELS DO

    fbVisionSourceB[uiVisionSource](
        Enable := GVL.g_aVisionTrackingSourceConfigB[uiVisionSource].Enable,
        Reset := GVL.g_xResetTrackingObjectSourceB,
        Config := GVL.g_aVisionTrackingSourceConfigB[uiVisionSource],
        Result := GVL.g_aVisionTrackingMultiResultB[uiVisionSource],
        ConveyorPositionMM := REAL_TO_LREAL(GVL.g_aConveyorRuntime[2].Status.PositionMM),
        Queue := GVL.g_stTrackingQueue_B
    );

END_FOR;

END_PROGRAM

// Just_Motion_Control_x86_64_Linux_SM_WV/Application/PRG_ROBOT/PRG_TrackingQueue_B
PROGRAM PRG_TrackingQueue_B
VAR
    uiObject : UINT; // Biến nội bộ uiObject.
    rCurrentConveyorPos : REAL; // Biến nội bộ rCurrentConveyorPos.
    rVelocityAbs : REAL; // Biến nội bộ rVelocityAbs.
    rDistanceToAbort : REAL; // Biến nội bộ rDistanceToAbort.
END_VAR

//=============================================================================
// PRG_TrackingQueue_A
//-----------------------------------------------------------------------------
// Cập nhật Runtime của tất cả Object trong Tracking Queue Robot B.
//
// Nguồn vị trí Conveyor:
//     GVL.g_aConveyorRuntime[2].Status.PositionMM
//
// Chương trình này KHÔNG tạo Object.
// Sensor/Vision Source sẽ chịu trách nhiệm tạo Object ở bước sau.
//=============================================================================

rCurrentConveyorPos := GVL.g_aConveyorRuntime[2].Status.PositionMM;
rVelocityAbs := ABS(GVL.g_aConveyorRuntime[2].Status.VelocityMMs);

//=============================================================================
// CLEAR TOÀN BỘ TRACKING QUEUE
//-----------------------------------------------------------------------------
IF GVL.g_xClearTrackingQueueB THEN

    FOR uiObject := 1 TO GVL.C_MAX_TRACK_OBJECTS DO
        GVL.g_stTrackingQueue_B.Objects[uiObject].Valid := FALSE;
        GVL.g_stTrackingQueue_B.Objects[uiObject].ObjectID := 0;
        GVL.g_stTrackingQueue_B.Objects[uiObject].ProductClassID := 0;
        GVL.g_stTrackingQueue_B.Objects[uiObject].Reserved := FALSE;
        GVL.g_stTrackingQueue_B.Objects[uiObject].ReservedToolID := 0;
        GVL.g_stTrackingQueue_B.Objects[uiObject].CanPick := FALSE;
        GVL.g_stTrackingQueue_B.Objects[uiObject].AbortRequired := FALSE;
        GVL.g_stTrackingQueue_B.Objects[uiObject].State := E_TrackingObjectState.OBJ_EMPTY;
        GVL.g_stTrackingQueue_B.Objects[uiObject].MissCode := 0;
        GVL.g_stTrackingQueue_B.Objects[uiObject].ErrorID := 0;
        GVL.g_stTrackingQueue_B.Objects[uiObject].TimeRemainingSec := 0.0;
        GVL.g_stTrackingQueue_B.Objects[uiObject].ConveyorOffset := 0.0;
        GVL.g_stTrackingQueue_B.Objects[uiObject].ConveyorCoordinate := 0.0;
    END_FOR;

    GVL.g_stTrackingQueue_B.ValidCount := 0;
    GVL.g_stTrackingQueue_B.ActiveIndex := GVL.C_INVALID_INDEX;

    // Nếu muốn ObjectID quay lại từ 1 sau mỗi lần clear.
    GVL.g_stTrackingQueue_B.NextObjectID := 0;

    // Tự hạ lệnh.
    GVL.g_xClearTrackingQueueB := FALSE;

    RETURN;
END_IF;


//=============================================================================
// DUYỆT TOÀN BỘ QUEUE
//=============================================================================
FOR uiObject := 1 TO GVL.C_MAX_TRACK_OBJECTS DO

    //----------------------------------------------------------------------
    // Chỉ xử lý Slot đang có Object hợp lệ.
    //----------------------------------------------------------------------
    IF GVL.g_stTrackingQueue_B.Objects[uiObject].Valid THEN

        //------------------------------------------------------------------
        // 1. CẬP NHẬT VỊ TRÍ CONVEYOR HIỆN TẠI
        //------------------------------------------------------------------
        GVL.g_stTrackingQueue_B.Objects[uiObject].CurrentConveyorPositionMM :=
            REAL_TO_LREAL(rCurrentConveyorPos);


        //------------------------------------------------------------------
        // 2. ĐỘ DỊCH CONVEYOR TỪ THỜI ĐIỂM CAPTURE
        //------------------------------------------------------------------
        GVL.g_stTrackingQueue_B.Objects[uiObject].ConveyorOffset :=
            LREAL_TO_REAL(
                GVL.g_stTrackingQueue_B.Objects[uiObject].CurrentConveyorPositionMM
                - GVL.g_stTrackingQueue_B.Objects[uiObject].CaptureConveyorPositionMM
            );


        //------------------------------------------------------------------
        // 3. TỌA ĐỘ DỌC CONVEYOR HIỆN TẠI CỦA OBJECT
        //------------------------------------------------------------------
        // PoseInConveyor.X là tọa độ Object tại thời điểm Capture.
        GVL.g_stTrackingQueue_B.Objects[uiObject].ConveyorCoordinate :=
            GVL.g_stTrackingQueue_B.Objects[uiObject].PoseInConveyor.X
            + GVL.g_stTrackingQueue_B.Objects[uiObject].ConveyorOffset;


        //------------------------------------------------------------------
        // 4. CURRENT POS
        //------------------------------------------------------------------
        GVL.g_stTrackingQueue_B.Objects[uiObject].CurrentPos :=
            GVL.g_stTrackingQueue_B.Objects[uiObject].PoseInConveyor;

        GVL.g_stTrackingQueue_B.Objects[uiObject].CurrentPos.X :=
            GVL.g_stTrackingQueue_B.Objects[uiObject].ConveyorCoordinate;


        //------------------------------------------------------------------
        // 5. DEFAULT RUNTIME FLAGS
        //------------------------------------------------------------------
//         GVL.g_stTrackingQueue_B.Objects[uiObject].CanPick := FALSE;
//         GVL.g_stTrackingQueue_B.Objects[uiObject].AbortRequired := FALSE;
        GVL.g_stTrackingQueue_B.Objects[uiObject].TimeRemainingSec := 0.0;


//         //------------------------------------------------------------------
// 		// DEFAULT RUNTIME FLAGS
// 		//------------------------------------------------------------------
// 		GVL.g_stTrackingQueue_B.Objects[uiObject].CanPick := FALSE;
// 		GVL.g_stTrackingQueue_B.Objects[uiObject].AbortRequired := FALSE;
		
		
		//----------------------------------------------------------------------
		// OBJECT ĐÃ PICK XONG
		// Không được tính lại READY/MISSED theo vị trí Conveyor.
		//----------------------------------------------------------------------
		IF GVL.g_stTrackingQueue_B.Objects[uiObject].State
			= E_TrackingObjectState.OBJ_PICKED THEN
		
			GVL.g_stTrackingQueue_B.Objects[uiObject].CanPick := FALSE;
			GVL.g_stTrackingQueue_B.Objects[uiObject].AbortRequired := FALSE;
		
		
		//----------------------------------------------------------------------
		// OBJECT CHƯA ĐƯỢC ROBOT / TOOL SỞ HỮU
		//----------------------------------------------------------------------
		ELSIF NOT GVL.g_stTrackingQueue_B.Objects[uiObject].Reserved THEN
		
			GVL.g_stTrackingQueue_B.Objects[uiObject].CanPick := FALSE;
			GVL.g_stTrackingQueue_B.Objects[uiObject].AbortRequired := FALSE;
		
			IF GVL.g_stTrackingQueue_B.Objects[uiObject].ConveyorCoordinate
				< GVL.g_stTrackingConfig_B.Workspace.PickZoneStartMM THEN
		
				GVL.g_stTrackingQueue_B.Objects[uiObject].State :=
					E_TrackingObjectState.OBJ_WAIT_PICK_ZONE;
		
			ELSIF GVL.g_stTrackingQueue_B.Objects[uiObject].ConveyorCoordinate
				<= GVL.g_stTrackingConfig_B.Workspace.PickZoneEndMM THEN
		
				GVL.g_stTrackingQueue_B.Objects[uiObject].CanPick := TRUE;
		
				GVL.g_stTrackingQueue_B.Objects[uiObject].State :=
					E_TrackingObjectState.OBJ_READY;
		
			ELSIF GVL.g_stTrackingQueue_B.Objects[uiObject].ConveyorCoordinate
				< GVL.g_stTrackingConfig_B.Workspace.ExpirePositionMM THEN
		
				GVL.g_stTrackingQueue_B.Objects[uiObject].State :=
					E_TrackingObjectState.OBJ_MISSED;
		
			ELSE
		
				GVL.g_stTrackingQueue_B.Objects[uiObject].State :=
					E_TrackingObjectState.OBJ_EXPIRED;
		
			END_IF;
		
		
		//----------------------------------------------------------------------
		// OBJECT ĐANG ĐƯỢC TRACKING SỞ HỮU
		//----------------------------------------------------------------------
		ELSE
		
			IF GVL.g_stTrackingQueue_B.Objects[uiObject].ConveyorCoordinate
				>= GVL.g_stTrackingConfig_B.Workspace.AbortPositionMM THEN
		
				GVL.g_stTrackingQueue_B.Objects[uiObject].AbortRequired := TRUE;
		
			ELSE
		
				GVL.g_stTrackingQueue_B.Objects[uiObject].AbortRequired := FALSE;
		
			END_IF;
		
		END_IF;
		
		
		//=============================================================================
		// CLEANUP OBJECT PICKED
		//=============================================================================
		IF GVL.g_stTrackingQueue_B.Objects[uiObject].Valid
		AND NOT GVL.g_stTrackingQueue_B.Objects[uiObject].Reserved
		AND GVL.g_stTrackingQueue_B.Objects[uiObject].State
			= E_TrackingObjectState.OBJ_PICKED THEN
		
			GVL.g_stTrackingQueue_B.Objects[uiObject].Valid := FALSE;
			GVL.g_stTrackingQueue_B.Objects[uiObject].ReservedToolID := 0;
			GVL.g_stTrackingQueue_B.Objects[uiObject].CanPick := FALSE;
			GVL.g_stTrackingQueue_B.Objects[uiObject].AbortRequired := FALSE;
			GVL.g_stTrackingQueue_B.Objects[uiObject].TimeRemainingSec := 0.0;
		
			GVL.g_stTrackingQueue_B.Objects[uiObject].State :=
				E_TrackingObjectState.OBJ_EMPTY;
		
			IF GVL.g_stTrackingQueue_B.ValidCount > 0 THEN
				GVL.g_stTrackingQueue_B.ValidCount :=
					GVL.g_stTrackingQueue_B.ValidCount - 1;
			END_IF;
		
		END_IF;



// 		//------------------------------------------------------------------
// 		// OBJECT CHƯA ĐƯỢC ROBOT / TOOL SỞ HỮU
// 		//------------------------------------------------------------------
// 		IF NOT GVL.g_stTrackingQueue_B.Objects[uiObject].Reserved THEN
// 		
// 			// Queue Manager được quyền tính lại hai trạng thái này.
// 			GVL.g_stTrackingQueue_B.Objects[uiObject].CanPick := FALSE;
// 			GVL.g_stTrackingQueue_B.Objects[uiObject].AbortRequired := FALSE;
// 		
// 			// Chưa tới vùng Pick.
// 			IF GVL.g_stTrackingQueue_B.Objects[uiObject].ConveyorCoordinate
// 				< GVL.g_stTrackingConfig_B.Workspace.PickZoneStartMM THEN
// 		
// 				GVL.g_stTrackingQueue_B.Objects[uiObject].State :=
// 					E_TrackingObjectState.OBJ_WAIT_PICK_ZONE;
// 		
// 			// Đang nằm trong vùng Pick.
// 			ELSIF GVL.g_stTrackingQueue_B.Objects[uiObject].ConveyorCoordinate
// 				<= GVL.g_stTrackingConfig_B.Workspace.PickZoneEndMM THEN
// 		
// 				GVL.g_stTrackingQueue_B.Objects[uiObject].CanPick := TRUE;
// 		
// 				GVL.g_stTrackingQueue_B.Objects[uiObject].State :=
// 					E_TrackingObjectState.OBJ_READY;
// 		
// 			// Đã ra khỏi vùng Pick nhưng chưa Expire.
// 			ELSIF GVL.g_stTrackingQueue_B.Objects[uiObject].ConveyorCoordinate
// 				< GVL.g_stTrackingConfig_B.Workspace.ExpirePositionMM THEN
// 		
// 				GVL.g_stTrackingQueue_B.Objects[uiObject].State :=
// 					E_TrackingObjectState.OBJ_MISSED;
// 		
// 			// Hết hiệu lực hoàn toàn.
// 			ELSE
// 		
// 				GVL.g_stTrackingQueue_B.Objects[uiObject].State :=
// 					E_TrackingObjectState.OBJ_EXPIRED;
// 		
// 			END_IF;
// 				
// 		
// 		//------------------------------------------------------------------
// 		// OBJECT ĐÃ ĐƯỢC ROBOT / TOOL SỞ HỮU
// 		//------------------------------------------------------------------
// 		ELSE
// 		
// 			// QUAN TRỌNG:
// 			// Không thay đổi CanPick tại đây.
// 			// Object đã được chọn khi CanPick = TRUE.
// 		
// 			// Chỉ tiếp tục theo dõi điều kiện Abort.
// 			IF GVL.g_stTrackingQueue_B.Objects[uiObject].ConveyorCoordinate
// 				>= GVL.g_stTrackingConfig_B.Workspace.AbortPositionMM THEN
// 		
// 				GVL.g_stTrackingQueue_B.Objects[uiObject].AbortRequired := TRUE;
// 		
// 			ELSE
// 		
// 				GVL.g_stTrackingQueue_B.Objects[uiObject].AbortRequired := FALSE;
// 		
// 			END_IF;
// 		
// 		END_IF;


        //------------------------------------------------------------------
        // 7. TÍNH THỜI GIAN CÒN LẠI TRƯỚC ABORT
        //------------------------------------------------------------------
        IF rVelocityAbs > 0.01 THEN

            rDistanceToAbort :=
                GVL.g_stTrackingConfig_B.Workspace.AbortPositionMM
                - GVL.g_stTrackingQueue_B.Objects[uiObject].ConveyorCoordinate;

            IF rDistanceToAbort > 0.0 THEN
                GVL.g_stTrackingQueue_B.Objects[uiObject].TimeRemainingSec :=
                    rDistanceToAbort / rVelocityAbs;
            ELSE
                GVL.g_stTrackingQueue_B.Objects[uiObject].TimeRemainingSec := 0.0;
            END_IF;

        END_IF;
		
		//=============================================================================
		// CLEANUP OBJECT ĐÃ EXPIRED
		//-----------------------------------------------------------------------------
		// Object đã ra khỏi toàn bộ vùng Tracking và không còn được Tool sở hữu.
		// Giải phóng Slot để Sensor có thể sử dụng lại.
		//=============================================================================
		IF NOT GVL.g_stTrackingQueue_B.Objects[uiObject].Reserved
		AND GVL.g_stTrackingQueue_B.Objects[uiObject].State = E_TrackingObjectState.OBJ_EXPIRED THEN
		
			// Giải phóng Object.
			GVL.g_stTrackingQueue_B.Objects[uiObject].Valid := FALSE;
			GVL.g_stTrackingQueue_B.Objects[uiObject].Reserved := FALSE;
			GVL.g_stTrackingQueue_B.Objects[uiObject].ReservedToolID := 0;
		
			// Xóa trạng thái runtime.
			GVL.g_stTrackingQueue_B.Objects[uiObject].CanPick := FALSE;
			GVL.g_stTrackingQueue_B.Objects[uiObject].AbortRequired := FALSE;
			GVL.g_stTrackingQueue_B.Objects[uiObject].TimeRemainingSec := 0.0;
		
			// Đưa Slot về Empty.
			GVL.g_stTrackingQueue_B.Objects[uiObject].State :=
				E_TrackingObjectState.OBJ_EMPTY;
		
			// Giảm số Object hợp lệ trong Queue.
			IF GVL.g_stTrackingQueue_B.ValidCount > 0 THEN
				GVL.g_stTrackingQueue_B.ValidCount :=
					GVL.g_stTrackingQueue_B.ValidCount - 1;
			END_IF;
		
		END_IF;

    END_IF;

END_FOR;

END_PROGRAM

// Just_Motion_Control_x86_64_Linux_SM_WV/Application/PRG_ROBOT/PRG_MultiToolTracking_B
PROGRAM PRG_MultiToolTracking_B
VAR
    fbControllerB : FB_MultiToolTrackingController_B;
    fbCoreInterfaceB : FB_TrackingCoreInterface_B;
    fbTrackingManagerB : FB_CONVEYOR_TRACKING_MANAGER_B;
    fbMotionAdapterB : FB_TrackingMotionQueueAdapter_B;
    fbSelectToolB : FB_SelectRobotTool_B;
    fbToolManagerB : ARRAY[0..GVL.C_MAX_TOOLS] OF FB_ToolManager_B;
    astToolCommandB : ARRAY[0..GVL.C_MAX_TOOLS] OF ST_ToolCommand;
    stCommandB : ST_MultiToolTrackingCommand;
    stConveyorOriginB : MC_COORD_REF;
    stFixedObjectPositionB : MC_COORD_REF;
    diVirtualEncoderB : DINT;
    uiTool : UINT;
    xTrackingRequestValid : BOOL;
    rtCreateTestObjectB : R_TRIG;
    xCoreRequestValid : BOOL;
    rtMultiTrackStartTestB : R_TRIG;
    xMultiTrackTestExecuteB : BOOL := FALSE;
    rtDebugCoreStartB : R_TRIG;
    rtDebugExecuteToCoreB : R_TRIG;
    rtDebugCoreRequestValidB : R_TRIG;
    udiDebugCoreStartCountB : UDINT;
    udiDebugExecuteToCoreCountB : UDINT;
    udiDebugCoreRequestCountB : UDINT;
    xDebugCoreStartLatchedB : BOOL;
    xDebugExecuteToCoreLatchedB : BOOL;
    xDebugCoreRequestLatchedB : BOOL;
    rConveyorVelocityPrevB : REAL;
    xConveyorRuntimeFirstScanB : BOOL := TRUE;
    fbPower : MC_Power;
    count_scan : INT;
    i_count : INT;
    udiv : INT;
    count_cal_max : INT;
    count_cal : INT;
    pulse_old : DINT;
    pulse_track : DINT;
    delta : REAL;
    rPulsePerScan : REAL;
    rFractionAcc : REAL;
    diBasePulse : DINT;
    diPulseThisScan : DINT;
    diSmoothCount : DINT;
END_VAR

IF GVL.X[8] THEN
	GVL.g_xResetTrackingObjectSourceA := TRUE;
	GVL.g_xMultiTrackResetTestB := TRUE;
	GVL.g_xClearTrackingQueueA := TRUE;
ELSE
	GVL.g_xResetTrackingObjectSourceA := FALSE;
	GVL.g_xMultiTrackResetTestB := FALSE;
	GVL.g_xClearTrackingQueueA := FALSE;
	
END_IF;

//GVL.g_axDIA[1] := GVL.X[20];


//=============================================================================
// MULTI-TOOL TRACKING TEST COMMAND
//-----------------------------------------------------------------------------
// Chỉ tạo dữ liệu Command một lần tại cạnh lên của Start Test.
// Sau này khi Interpreter hoạt động, phần này chỉ dùng cho Commissioning/Test.
//=============================================================================

rtMultiTrackStartTestB(CLK := GVL.g_xMultiTrackStartTestB);
IF rtMultiTrackStartTestB.Q THEN
    GVL.g_stMultiTrackCommandB.CommandID := GVL.g_stMultiTrackCommandB.CommandID + 1;

    IF GVL.g_stMultiTrackCommandB.CommandID = 0 THEN
        GVL.g_stMultiTrackCommandB.CommandID := 1;
    END_IF;

//     GVL.g_stMultiTrackCommandB.RecipeID := 1;
//     GVL.g_stMultiTrackCommandB.TargetPickCountOverride := 1;
//     GVL.g_stMultiTrackCommandB.ToolMaskOverride := DWORD#1;
// 
//     GVL.g_aMultiTrackRecipeB[1].Enable := TRUE;
//     GVL.g_aMultiTrackRecipeB[1].RecipeID := 1;
//     GVL.g_aMultiTrackRecipeB[1].ProductClassID := 0;
//     GVL.g_aMultiTrackRecipeB[1].TargetPickCount := 1;
//     GVL.g_aMultiTrackRecipeB[1].ToolEnableMask := DWORD#1;

	GVL.g_stMultiTrackCommandB.RecipeID := 1;
    GVL.g_stMultiTrackCommandB.TargetPickCountOverride := 1;
    GVL.g_stMultiTrackCommandB.ToolMaskOverride := DWORD#1;

    GVL.g_aMultiTrackRecipeB[1].Enable := TRUE;
    GVL.g_aMultiTrackRecipeB[1].RecipeID := 1;
    GVL.g_aMultiTrackRecipeB[1].ProductClassID := 0;
    GVL.g_aMultiTrackRecipeB[1].TargetPickCount := 1;
    GVL.g_aMultiTrackRecipeB[1].ToolEnableMask := DWORD#1;

    xMultiTrackTestExecuteB := TRUE;
END_IF;

// Khi Controller hoàn thành hoặc lỗi thì hạ Execute test.
IF GVL.g_stMultiTrackStatusB.Done OR GVL.g_stMultiTrackStatusB.Error OR GVL.g_xMultiTrackResetTestB OR GVL.g_xMultiTrackAbortTestB THEN
    xMultiTrackTestExecuteB := FALSE;
END_IF;

stCommandB := GVL.g_stMultiTrackCommandB;

stCommandB.Execute := GVL.g_stMultiTrackCommandB.Execute OR xMultiTrackTestExecuteB;

stCommandB.Reset := GVL.g_stMultiTrackCommandB.Reset OR GVL.g_xMultiTrackResetTestB;

stCommandB.Abort :=
    GVL.g_stMultiTrackCommandB.Abort
    OR GVL.g_xMultiTrackAbortTestB;


//=============================================================================
// 02. GỐC CONVEYOR VÀ OBJECT TEST
//-----------------------------------------------------------------------------
// Sau này thay stConveyorOriginB bằng cấu hình Conveyor thực tế trên HMI.
//=============================================================================
// stConveyorOriginB.X := 350.0;
// stConveyorOriginB.Y := -200.0;
// stConveyorOriginB.Z := 150.0;
// stConveyorOriginB.A := 90.0;
// stConveyorOriginB.B := 0.0;
// stConveyorOriginB.C := 0.0;

stConveyorOriginB.X := GVL.g_aConveyorRuntime[2].Config.Origin.X;
stConveyorOriginB.Y := GVL.g_aConveyorRuntime[2].Config.Origin.Y;
stConveyorOriginB.Z := GVL.g_aConveyorRuntime[2].Config.Origin.Z;
stConveyorOriginB.A := GVL.g_aConveyorRuntime[2].Config.Origin.A;
stConveyorOriginB.B := 0.0;
stConveyorOriginB.C := 0.0;

stFixedObjectPositionB := GVL.g_stTrackingSimulation.FixedObjectPosition;

// Power Axis 6
fbPower(
    Axis := AXIS_5,
    Enable := TRUE,
    bRegulatorOn := TRUE,
    bDriveStart := TRUE
);
i_count := 100;
count_cal_max := 3;
IF GVL.Y[11] <> FALSE  THEN
	IF count_scan = 0 THEN
		pulse_old := AXIS_5.diActPosition;
	END_IF
	count_scan := count_scan + 1;
	
	IF count_scan >= i_count THEN
		rPulsePerScan := TO_REAL((AXIS_5.diActPosition - pulse_old))/(i_count);
		GVL.g_HMI_PulsePerCycle_Cr := rPulsePerScan;
		count_scan := 0;
		count_cal := count_cal + 1;
	END_IF
END_IF;
udiv := udiv + 1;


IF count_cal >= count_cal_max THEN
	// Phần nguyên.
	diBasePulse := REAL_TO_DINT(TRUNC(rPulsePerScan));
	
	// Tích lũy phần lẻ.
	rFractionAcc := rFractionAcc + (rPulsePerScan - DINT_TO_REAL(diBasePulse));
	
	// Mặc định chỉ tăng phần nguyên.
	diPulseThisScan := diBasePulse;
	
	// Khi phần lẻ tích đủ 1 xung thì bù thêm 1.
	IF rFractionAcc <= -200.0 THEN
		diPulseThisScan := diPulseThisScan - 1;
		rFractionAcc := rFractionAcc + 1.0;
	END_IF;
	
	// Position đưa sang encoder trung gian.
	IF GVL.Y[11] <> FALSE THEN
		diSmoothCount := diSmoothCount + diPulseThisScan;
	END_IF
END_IF


//=============================================================================
// 03. ENCODER ẢO
//-----------------------------------------------------------------------------
// Phần này được chuyển từ PRG_ConveyorTracking cũ sang PRG mới.
//=============================================================================
IF GVL.g_stTrackingSimulation.VirtualEncoderReset THEN
    diVirtualEncoderB := 0;
ELSIF GVL.g_stTrackingSimulation.VirtualEncoderEnable THEN
    diVirtualEncoderB := diVirtualEncoderB + GVL.g_stTrackingSimulation.VirtualEncoderStepPerCycle;
END_IF;

IF GVL.g_stTrackingSimulation.Mode <> E_ApplicationSimulationMode.SIM_OFF AND GVL.g_stTrackingSimulation.VirtualEncoderEnable THEN 
	SMC_FreeEncoder_B.diEncoderPosition := diVirtualEncoderB; 
ELSE
	//SMC_FreeEncoder_B.diEncoderPosition := TO_DINT(AXIS_6_B.fActPosition);
	//SMC_FreeEncoder_B.diEncoderPosition :=AXIS_6_B.diActPosition;
// 	IF udiv < 400 THEN
// 		SMC_FreeEncoder_B.diEncoderPosition := SMC_FreeEncoder_B.diEncoderPosition - 10;
// 	END_IF
// 	IF udiv >= 400 THEN
// 		SMC_FreeEncoder_B.diEncoderPosition := SMC_FreeEncoder_B.diEncoderPosition - 11;
// 	END_IF
// 	IF udiv = 3 THEN
// 		SMC_FreeEncoder_B.diEncoderPosition := SMC_FreeEncoder_B.diEncoderPosition - 5;
// 	END_IF
// 	IF udiv = 4 THEN
// 		SMC_FreeEncoder_B.diEncoderPosition := SMC_FreeEncoder_B.diEncoderPosition - 5;
// 	END_IF
	IF GVL.Y[11] <> FALSE THEN
		SMC_FreeEncoder_B.diEncoderPosition := SMC_FreeEncoder_B.diEncoderPosition - GVL.g_HMI_PulsePerCycle_Set_B;
	END_IF;
END_IF;

IF udiv = 800 THEN udiv := 0; END_IF;
//=============================================================================
// 04. CONVEYOR RUNTIME STATUS
//-----------------------------------------------------------------------------
// Logical Axis SM_Drive_Logical_B đã được scale:
//     fActPosition = mm
//     fActVelocity = mm/s
//
// Mục đích:
//     - Cập nhật Status cho HMI.
//     - Làm nguồn dữ liệu chung cho Queue/Sensor/Vision.
//     - Tracking Manager đọc cùng một nguồn trạng thái Conveyor.
//=============================================================================

//-----------------------------------------------------------------------------
// 1. RAW POSITION / VELOCITY
//-----------------------------------------------------------------------------
GVL.g_aConveyorRuntime[2].Status.RawPosition :=
    LREAL_TO_REAL(SM_Drive_Logical_B.fActPosition);

GVL.g_aConveyorRuntime[2].Status.RawVelocity :=
    LREAL_TO_REAL(SM_Drive_Logical_B.fActVelocity);


//-----------------------------------------------------------------------------
// 2. POSITION THEO CHIỀU QUY ƯỚC CỦA APPLICATION
//-----------------------------------------------------------------------------
// DirectionSign:
//      +1 = giữ nguyên chiều Axis.
//      -1 = đảo chiều quy ước.
IF GVL.g_aConveyorRuntime[2].Config.DirectionSign >= 0 THEN
    GVL.g_aConveyorRuntime[2].Status.PositionMM :=
        LREAL_TO_REAL(SM_Drive_Logical_B.fActPosition);
ELSE
    GVL.g_aConveyorRuntime[2].Status.PositionMM :=
        -LREAL_TO_REAL(SM_Drive_Logical_B.fActPosition);
END_IF;


//-----------------------------------------------------------------------------
// 3. VELOCITY THEO CHIỀU QUY ƯỚC
//-----------------------------------------------------------------------------
IF GVL.g_aConveyorRuntime[2].Config.DirectionSign >= 0 THEN
    GVL.g_aConveyorRuntime[2].Status.VelocityMMs :=
        LREAL_TO_REAL(SM_Drive_Logical_B.fActVelocity);
ELSE
    GVL.g_aConveyorRuntime[2].Status.VelocityMMs :=
        -LREAL_TO_REAL(SM_Drive_Logical_B.fActVelocity);
END_IF;


//-----------------------------------------------------------------------------
// 4. GIỚI HẠN FILTER FACTOR 0.0 ... 1.0
//-----------------------------------------------------------------------------
IF GVL.g_aConveyorRuntime[2].Config.VelocityFilterFactor < 0.0 THEN
    GVL.g_aConveyorRuntime[2].Config.VelocityFilterFactor := 0.0;
ELSIF GVL.g_aConveyorRuntime[2].Config.VelocityFilterFactor > 1.0 THEN
    GVL.g_aConveyorRuntime[2].Config.VelocityFilterFactor := 1.0;
END_IF;


//-----------------------------------------------------------------------------
// 5. LOW-PASS FILTER VELOCITY
//-----------------------------------------------------------------------------
// FilterFactor = 1.0 : gần như lấy trực tiếp Velocity.
// FilterFactor nhỏ   : lọc mượt hơn nhưng phản ứng chậm hơn.
GVL.g_aConveyorRuntime[2].Status.FilteredVelocityMMs :=
    GVL.g_aConveyorRuntime[2].Status.FilteredVelocityMMs
    + GVL.g_aConveyorRuntime[2].Config.VelocityFilterFactor
    * (
        GVL.g_aConveyorRuntime[2].Status.VelocityMMs
        - GVL.g_aConveyorRuntime[2].Status.FilteredVelocityMMs
    );


//-----------------------------------------------------------------------------
// 6. ACCELERATION
//-----------------------------------------------------------------------------
// PRG_MultiToolTracking_A hiện chạy trong task 4 ms.
// a = Delta V / 0.004 s.
IF xConveyorRuntimeFirstScanB THEN

    GVL.g_aConveyorRuntime[2].Status.AccelerationMMs2 := 0.0;

    rConveyorVelocityPrevB :=
        GVL.g_aConveyorRuntime[2].Status.FilteredVelocityMMs;

    xConveyorRuntimeFirstScanB := FALSE;

ELSE

    GVL.g_aConveyorRuntime[2].Status.AccelerationMMs2 :=
        (
            GVL.g_aConveyorRuntime[2].Status.FilteredVelocityMMs
            - rConveyorVelocityPrevB
        ) / 0.004;

    rConveyorVelocityPrevB :=
        GVL.g_aConveyorRuntime[2].Status.FilteredVelocityMMs;

END_IF;


//-----------------------------------------------------------------------------
// 7. RUNNING / STANDSTILL / DIRECTION
//-----------------------------------------------------------------------------
IF ABS(GVL.g_aConveyorRuntime[2].Status.FilteredVelocityMMs)
    > GVL.g_aConveyorRuntime[2].Config.RunningThresholdMMs THEN

    GVL.g_aConveyorRuntime[2].Status.Running := TRUE;
    GVL.g_aConveyorRuntime[2].Status.Standstill := FALSE;

    IF GVL.g_aConveyorRuntime[2].Status.FilteredVelocityMMs > 0.0 THEN
        GVL.g_aConveyorRuntime[2].Status.Direction := 1;
    ELSE
        GVL.g_aConveyorRuntime[2].Status.Direction := -1;
    END_IF;

ELSE

    GVL.g_aConveyorRuntime[2].Status.Running := FALSE;
    GVL.g_aConveyorRuntime[2].Status.Standstill := TRUE;
    GVL.g_aConveyorRuntime[2].Status.Direction := 0;

END_IF;


//-----------------------------------------------------------------------------
// 8. VALID
//-----------------------------------------------------------------------------
GVL.g_aConveyorRuntime[2].Status.Valid :=
    GVL.g_aConveyorRuntime[2].Config.Enable;


//-----------------------------------------------------------------------------
// 9. ERROR LIMIT CHECK
//-----------------------------------------------------------------------------
GVL.g_aConveyorRuntime[2].Status.Error := FALSE;
GVL.g_aConveyorRuntime[2].Status.ErrorID := 0;

IF GVL.g_aConveyorRuntime[2].Config.MaxVelocityMMs > 0.0
AND ABS(GVL.g_aConveyorRuntime[2].Status.VelocityMMs)
    > GVL.g_aConveyorRuntime[2].Config.MaxVelocityMMs THEN

    GVL.g_aConveyorRuntime[2].Status.Error := TRUE;
    GVL.g_aConveyorRuntime[2].Status.ErrorID := 9001;

ELSIF GVL.g_aConveyorRuntime[2].Config.MaxAccelerationMMs2 > 0.0
AND ABS(GVL.g_aConveyorRuntime[2].Status.AccelerationMMs2)
    > GVL.g_aConveyorRuntime[2].Config.MaxAccelerationMMs2 THEN

    GVL.g_aConveyorRuntime[2].Status.Error := TRUE;
    GVL.g_aConveyorRuntime[2].Status.ErrorID := 9002;

END_IF;


rtCreateTestObjectB(CLK := GVL.g_xCreateTestTrackingObjectB);

IF rtCreateTestObjectB.Q THEN
    GVL.g_stTrackingQueue_B.NextObjectID := GVL.g_stTrackingQueue_B.NextObjectID + 1;
    IF GVL.g_stTrackingQueue_B.NextObjectID = 0 THEN GVL.g_stTrackingQueue_B.NextObjectID := 1; END_IF;

    GVL.g_stTrackingQueue_B.Objects[1].Valid := TRUE;
    GVL.g_stTrackingQueue_B.Objects[1].ObjectID := GVL.g_stTrackingQueue_B.NextObjectID;
    GVL.g_stTrackingQueue_B.Objects[1].ProductClassID := 1;
    GVL.g_stTrackingQueue_B.Objects[1].Reserved := FALSE;
    GVL.g_stTrackingQueue_B.Objects[1].ReservedToolID := 0;
    GVL.g_stTrackingQueue_B.Objects[1].CanPick := TRUE;
    GVL.g_stTrackingQueue_B.Objects[1].OrientationValid := TRUE;
    GVL.g_stTrackingQueue_B.Objects[1].VisionScore := 100.0;
    GVL.g_stTrackingQueue_B.Objects[1].State := E_TrackingObjectState.OBJ_READY;

    GVL.g_stTrackingQueue_B.Objects[1].VisionPos.X := 000.0;
    GVL.g_stTrackingQueue_B.Objects[1].VisionPos.Y := 0.0;
    GVL.g_stTrackingQueue_B.Objects[1].VisionPos.Z := 50.0;
    GVL.g_stTrackingQueue_B.Objects[1].VisionPos.A := 0.0;
	
	//-------------------------------------------------------------------------
	// OBJECT 1 - POSE CHUẨN TRONG HỆ CONVEYOR
	//-------------------------------------------------------------------------
	GVL.g_stTrackingQueue_B.Objects[1].PoseInConveyor.X := 000.0;
	GVL.g_stTrackingQueue_B.Objects[1].PoseInConveyor.Y := 0.0;
	GVL.g_stTrackingQueue_B.Objects[1].PoseInConveyor.Z := 50.0;
	GVL.g_stTrackingQueue_B.Objects[1].PoseInConveyor.A := 0.0;

	
	// Chốt vị trí Conveyor đúng thời điểm Object được tạo.
	GVL.g_stTrackingQueue_B.Objects[1].CaptureConveyorPositionMM :=
		REAL_TO_LREAL(GVL.g_aConveyorRuntime[2].Status.PositionMM);
	
	//---------------------------------------------------------------------
    // OBJECT 2
    //---------------------------------------------------------------------
    GVL.g_stTrackingQueue_B.NextObjectID :=
        GVL.g_stTrackingQueue_B.NextObjectID + 1;

    IF GVL.g_stTrackingQueue_B.NextObjectID = 0 THEN
        GVL.g_stTrackingQueue_B.NextObjectID := 1;
    END_IF;

